LIN {X 0,Y 297.522,Z 437.012,A -85,B 0,C 180,E1 -16370.483,E2 -16370.483} C_VEL
LIN {X 0,Y 297.104,Z 437.216,A -85,B 0,C 180,E1 -16373.208,E2 -16373.208} C_VEL
LIN {X 0,Y 296.911,Z 436.192,A -85,B 0,C 180,E1 -16375.928,E2 -16375.928} C_VEL
LIN {X 0,Y 296.872,Z 433.944,A -85,B 0,C 180,E1 -16378.644,E2 -16378.644} C_VEL
LIN {X 0,Y 296.926,Z 430.435,A -85,B 0,C 180,E1 -16381.357,E2 -16381.357} C_VEL
LIN {X 0,Y 297.311,Z 426.96,A -85,B 0,C 180,E1 -16383.388,E2 -16383.388} C_VEL
LIN {X 0,Y 297.857,Z 421.058,A -85,B 0,C 180,E1 -16386.095,E2 -16386.095} C_VEL
LIN {X 0,Y 298.455,Z 414.521,A -85,B 0,C 180,E1 -16388.499,E2 -16388.499} C_VEL
LIN {X 0,Y 299.541,Z 405.637,A -85,B 0,C 180,E1 -16391.161,E2 -16391.161} C_VEL
LIN {X 0,Y 300.946,Z 396.119,A -85,B 0,C 180,E1 -16393.505,E2 -16393.505} C_VEL
LIN {X 0,Y 302.502,Z 384.733,A -85,B 0,C 180,E1 -16395.842,E2 -16395.842} C_VEL
LIN {X 0,Y 304.428,Z 372.118,A -85,B 0,C 180,E1 -16397.986,E2 -16397.986} C_VEL
LIN {X 0,Y 306.235,Z 358.613,A -85,B 0,C 180,E1 -16399.902,E2 -16399.902} C_VEL
LIN {X 0,Y 308.168,Z 344.283,A -85,B 0,C 180,E1 -16401.577,E2 -16401.577} C_VEL
LIN {X 0,Y 309.992,Z 329.479,A -85,B 0,C 180,E1 -16402.99,E2 -16402.99} C_VEL
LIN {X 0,Y 309.934,Z 327.134,A -85,B 0,C 180,E1 -16403.209,E2 -16403.209} C_VEL
LIN {X 0,Y 306.166,Z 312.141,A -85,B 0,C 180,E1 -16404.665,E2 -16404.665} C_VEL
LIN {X 0,Y 301.591,Z 296.002,A -85,B 0,C 180,E1 -16406.023,E2 -16406.023} C_VEL
LIN {X 0,Y 297.601,Z 283.041,A -85,B 0,C 180,E1 -16407.007,E2 -16407.007} C_VEL
LIN {X 0,Y 297.87,Z 283.005,A -85,B 0,C 180,E1 -16409.702,E2 -16409.702} C_VEL
LIN {X 0,Y 298.165,Z 282.969,A -85,B 0,C 180,E1 -16412.829,E2 -16412.829} C_VEL
LIN {X 0,Y 298.368,Z 282.942,A -85,B 0,C 180,E1 -16416.077,E2 -16416.077} C_VEL
LIN {X 0,Y 298.403,Z 282.94,A -85,B 0,C 180,E1 -16419.488,E2 -16419.488} C_VEL
LIN {X 0,Y 298.401,Z 282.942,A -85,B 0,C 180,E1 -16423.103,E2 -16423.103} C_VEL
LIN {X 0,Y 298.405,Z 282.941,A -85,B 0,C 180,E1 -16426.921,E2 -16426.921} C_VEL
LIN {X 0,Y 298.401,Z 282.941,A -85,B 0,C 180,E1 -16431.007,E2 -16431.007} C_VEL
LIN {X 0,Y 298.421,Z 282.935,A -85,B 0,C 180,E1 -16433.93,E2 -16433.93} C_VEL
LIN {X 0,Y 298.396,Z 282.938,A -85,B 0,C 180,E1 -16437.984,E2 -16437.984} C_VEL
LIN {X 0,Y 298.46,Z 282.93,A -85,B 0,C 180,E1 -16441.904,E2 -16441.904} C_VEL
LIN {X 0,Y 298.484,Z 282.928,A -85,B 0,C 180,E1 -16444.924,E2 -16444.924} C_VEL
LIN {X 0,Y 298.436,Z 282.933,A -85,B 0,C 180,E1 -16449.314,E2 -16449.314} C_VEL
LIN {X 0,Y 298.538,Z 282.924,A -85,B 0,C 180,E1 -16452.179,E2 -16452.179} C_VEL
LIN {X 0,Y 298.597,Z 282.913,A -85,B 0,C 180,E1 -16454.995,E2 -16454.995} C_VEL
LIN {X 0,Y 298.594,Z 282.913,A -85,B 0,C 180,E1 -16459.147,E2 -16459.147} C_VEL
LIN {X 0,Y 298.701,Z 282.902,A -85,B 0,C 180,E1 -16461.884,E2 -16461.884} C_VEL
LIN {X 0,Y 298.637,Z 282.909,A -85,B 0,C 180,E1 -16464.599,E2 -16464.599} C_VEL
LIN {X 0,Y 298.923,Z 282.872,A -85,B 0,C 180,E1 -16468.653,E2 -16468.653} C_VEL
LIN {X 0,Y 298.922,Z 282.872,A -85,B 0,C 180,E1 -16471.347,E2 -16471.347} C_VEL
LIN {X 0,Y 298.643,Z 282.909,A -85,B 0,C 180,E1 -16475.401,E2 -16475.401} C_VEL
LIN {X 0,Y 298.713,Z 282.9,A -85,B 0,C 180,E1 -16478.115,E2 -16478.115} C_VEL
LIN {X 0,Y 298.553,Z 282.919,A -85,B 0,C 180,E1 -16482.232,E2 -16482.232} C_VEL
LIN {X 0,Y 298.609,Z 282.913,A -85,B 0,C 180,E1 -16485.209,E2 -16485.209} C_VEL
LIN {X 0,Y 298.543,Z 282.921,A -85,B 0,C 180,E1 -16489.243,E2 -16489.243} C_VEL
LIN {X 0,Y 298.461,Z 282.933,A -85,B 0,C 180,E1 -16493.598,E2 -16493.598} C_VEL
LIN {X 0,Y 298.488,Z 282.926,A -85,B 0,C 180,E1 -16496.575,E2 -16496.575} C_VEL
LIN {X 0,Y 298.42,Z 282.937,A -85,B 0,C 180,E1 -16499.641,E2 -16499.641} C_VEL
LIN {X 0,Y 298.398,Z 282.939,A -85,B 0,C 180,E1 -16502.8,E2 -16502.8} C_VEL
LIN {X 0,Y 298.431,Z 282.935,A -85,B 0,C 180,E1 -16506.803,E2 -16506.803} C_VEL
LIN {X 0,Y 298.376,Z 282.942,A -85,B 0,C 180,E1 -16509.492,E2 -16509.492} C_VEL
LIN {X 0,Y 298.374,Z 282.945,A -85,B 0,C 180,E1 -16513.097,E2 -16513.097} C_VEL
LIN {X 0,Y 298.406,Z 282.942,A -85,B 0,C 180,E1 -16516.921,E2 -16516.921} C_VEL
LIN {X 0,Y 298.402,Z 282.94,A -85,B 0,C 180,E1 -16521.007,E2 -16521.007} C_VEL
LIN {X 0,Y 298.421,Z 282.935,A -85,B 0,C 180,E1 -16523.93,E2 -16523.93} C_VEL
LIN {X 0,Y 298.397,Z 282.938,A -85,B 0,C 180,E1 -16527.984,E2 -16527.984} C_VEL
LIN {X 0,Y 298.461,Z 282.93,A -85,B 0,C 180,E1 -16531.904,E2 -16531.904} C_VEL
LIN {X 0,Y 298.485,Z 282.928,A -85,B 0,C 180,E1 -16534.924,E2 -16534.924} C_VEL
LIN {X 0,Y 298.444,Z 282.932,A -85,B 0,C 180,E1 -16539.314,E2 -16539.314} C_VEL
LIN {X 0,Y 298.542,Z 282.923,A -85,B 0,C 180,E1 -16542.179,E2 -16542.179} C_VEL
LIN {X 0,Y 298.597,Z 282.912,A -85,B 0,C 180,E1 -16544.995,E2 -16544.995} C_VEL
LIN {X 0,Y 298.587,Z 282.914,A -85,B 0,C 180,E1 -16549.146,E2 -16549.146} C_VEL
LIN {X 0,Y 298.702,Z 282.902,A -85,B 0,C 180,E1 -16551.884,E2 -16551.884} C_VEL
LIN {X 0,Y 298.639,Z 282.909,A -85,B 0,C 180,E1 -16554.598,E2 -16554.598} C_VEL
LIN {X 0,Y 298.924,Z 282.873,A -85,B 0,C 180,E1 -16558.652,E2 -16558.652} C_VEL
LIN {X 0,Y 298.922,Z 282.872,A -85,B 0,C 180,E1 -16561.347,E2 -16561.347} C_VEL
LIN {X 0,Y 298.854,Z 282.878,A -85,B 0,C 180,E1 -16562.103,E2 -16562.103} C_VEL
LIN {X 0,Y 298.135,Z 282.971,A -85,B 0,C 180,E1 -16563.226,E2 -16563.226} C_VEL
LIN {X 0,Y 295.21,Z 283.335,A -85,B 0,C 180,E1 -16565.053,E2 -16565.053} C_VEL
LIN {X 0,Y 292.761,Z 283.64,A -85,B 0,C 180,E1 -16566.536,E2 -16566.536} C_VEL
LIN {X 0,Y 291.726,Z 283.772,A -85,B 0,C 180,E1 -16567.686,E2 -16567.686} C_VEL
LIN {X 0,Y 291.649,Z 283.777,A -85,B 0,C 180,E1 -16568.075,E2 -16568.075} C_VEL
LIN {X 0,Y 291.521,Z 283.794,A -85,B 0,C 180,E1 -16572.531,E2 -16572.531} C_VEL
LIN {X 0,Y 291.558,Z 283.792,A -85,B 0,C 180,E1 -16575.376,E2 -16575.376} C_VEL
LIN {X 0,Y 291.453,Z 283.805,A -85,B 0,C 180,E1 -16579.874,E2 -16579.874} C_VEL
LIN {X 0,Y 291.366,Z 283.815,A -85,B 0,C 180,E1 -16584.208,E2 -16584.208} C_VEL
LIN {X 0,Y 291.355,Z 283.819,A -85,B 0,C 180,E1 -16587.278,E2 -16587.278} C_VEL
LIN {X 0,Y 291.391,Z 283.877,A -85,B 0,C 180,E1 -16589.079,E2 -16589.079} C_VEL
LIN {X 0,Y 291.971,Z 287.579,A -85,B 0,C 180,E1 -16592.596,E2 -16592.596} C_VEL
LIN {X 0,Y 292.796,Z 292.36,A -85,B 0,C 180,E1 -16596.875,E2 -16596.875} C_VEL
LIN {X 0,Y 293.772,Z 297.435,A -85,B 0,C 180,E1 -16601.139,E2 -16601.139} C_VEL
LIN {X 0,Y 294.512,Z 301.385,A -85,B 0,C 180,E1 -16604.283,E2 -16604.283} C_VEL
LIN {X 0,Y 294.887,Z 304.002,A -85,B 0,C 180,E1 -16606.278,E2 -16606.278} C_VEL
LIN {X 0,Y 294.882,Z 306.534,A -85,B 0,C 180,E1 -16608.138,E2 -16608.138} C_VEL
LIN {X 0,Y 294.127,Z 311.482,A -85,B 0,C 180,E1 -16611.592,E2 -16611.592} C_VEL
LIN {X 0,Y 293.063,Z 317.71,A -85,B 0,C 180,E1 -16615.796,E2 -16615.796} C_VEL
LIN {X 0,Y 297.438,Z 336.476,A -85,B 0,C 180,E1 -16617.196,E2 -16617.196} C_VEL
LIN {X 0,Y 300.916,Z 353.108,A -85,B 0,C 180,E1 -16618.669,E2 -16618.669} C_VEL
LIN {X 0,Y 303.835,Z 368.951,A -85,B 0,C 180,E1 -16620.322,E2 -16620.322} C_VEL
LIN {X 0,Y 305.212,Z 379.329,A -85,B 0,C 180,E1 -16621.521,E2 -16621.521} C_VEL
LIN {X 0,Y 302.653,Z 392.931,A -85,B 0,C 180,E1 -16623.075,E2 -16623.075} C_VEL
LIN {X 0,Y 300.081,Z 405.907,A -85,B 0,C 180,E1 -16624.881,E2 -16624.881} C_VEL
LIN {X 0,Y 297.678,Z 417.982,A -85,B 0,C 180,E1 -16626.913,E2 -16626.913} C_VEL
LIN {X 0,Y 295.517,Z 428.788,A -85,B 0,C 180,E1 -16629.1,E2 -16629.1} C_VEL
LIN {X 0,Y 293.557,Z 438.678,A -85,B 0,C 180,E1 -16631.505,E2 -16631.505} C_VEL
LIN {X 0,Y 292.031,Z 447.172,A -85,B 0,C 180,E1 -16634.005,E2 -16634.005} C_VEL
LIN {X 0,Y 290.853,Z 454.729,A -85,B 0,C 180,E1 -16636.729,E2 -16636.729} C_VEL
LIN {X 0,Y 290.093,Z 460.885,A -85,B 0,C 180,E1 -16639.531,E2 -16639.531} C_VEL
LIN {X 0,Y 289.749,Z 465.59,A -85,B 0,C 180,E1 -16642.333,E2 -16642.333} C_VEL
LIN {X 0,Y 289.648,Z 468.242,A -85,B 0,C 180,E1 -16644.43,E2 -16644.43} C_VEL
LIN {X 0,Y 289.543,Z 470.632,A -85,B 0,C 180,E1 -16647.217,E2 -16647.217} C_VEL
LIN {X 0,Y 289.657,Z 471.738,A -85,B 0,C 180,E1 -16650,E2 -16650} C_VEL
LIN {X 0,Y 289.539,Z 471.604,A -85,B 0,C 180,E1 -16652.783,E2 -16652.783} C_VEL
LIN {X 0,Y 289.585,Z 470.189,A -85,B 0,C 180,E1 -16655.712,E2 -16655.712} C_VEL
LIN {X 0,Y 289.712,Z 467.815,A -85,B 0,C 180,E1 -16658.369,E2 -16658.369} C_VEL
LIN {X 0,Y 290.177,Z 464.167,A -85,B 0,C 180,E1 -16661.172,E2 -16661.172} C_VEL
LIN {X 0,Y 291.19,Z 459.315,A -85,B 0,C 180,E1 -16663.967,E2 -16663.967} C_VEL
LIN {X 0,Y 292.734,Z 453.256,A -85,B 0,C 180,E1 -16666.744,E2 -16666.744} C_VEL
LIN {X 0,Y 295.205,Z 444.929,A -85,B 0,C 180,E1 -16669.831,E2 -16669.831} C_VEL
LIN {X 0,Y 298.479,Z 434.898,A -85,B 0,C 180,E1 -16672.862,E2 -16672.862} C_VEL
LIN {X 0,Y 302.294,Z 424.35,A -85,B 0,C 180,E1 -16675.474,E2 -16675.474} C_VEL
LIN {X 0,Y 306.87,Z 412.141,A -85,B 0,C 180,E1 -16678.002,E2 -16678.002} C_VEL
LIN {X 0,Y 311.549,Z 399.815,A -85,B 0,C 180,E1 -16680.127,E2 -16680.127} C_VEL
LIN {X 0,Y 316.135,Z 387.773,A -85,B 0,C 180,E1 -16681.878,E2 -16681.878} C_VEL
LIN {X 0,Y 318.826,Z 373.737,A -85,B 0,C 180,E1 -16684.272,E2 -16684.272} C_VEL
LIN {X 0,Y 319.606,Z 365.662,A -85,B 0,C 180,E1 -16685.875,E2 -16685.875} C_VEL
LIN {X 0,Y 319.866,Z 359.589,A -85,B 0,C 180,E1 -16687.285,E2 -16687.285} C_VEL
LIN {X 0,Y 319.968,Z 353.405,A -85,B 0,C 180,E1 -16689.036,E2 -16689.036} C_VEL
LIN {X 0,Y 320.152,Z 347.624,A -85,B 0,C 180,E1 -16691.191,E2 -16691.191} C_VEL
LIN {X 0,Y 320.329,Z 344.817,A -85,B 0,C 180,E1 -16692.855,E2 -16692.855} C_VEL
LIN {X 0,Y 320.856,Z 342.981,A -85,B 0,C 180,E1 -16694.502,E2 -16694.502} C_VEL
LIN {X 0,Y 321.371,Z 342.809,A -85,B 0,C 180,E1 -16696.193,E2 -16696.193} C_VEL
LIN {X 0,Y 322.187,Z 343.704,A -85,B 0,C 180,E1 -16697.873,E2 -16697.873} C_VEL
LIN {X 0,Y 323.235,Z 345.85,A -85,B 0,C 180,E1 -16699.552,E2 -16699.552} C_VEL
LIN {X 0,Y 324.353,Z 349.259,A -85,B 0,C 180,E1 -16701.265,E2 -16701.265} C_VEL
LIN {X 0,Y 325.411,Z 354.292,A -85,B 0,C 180,E1 -16703.045,E2 -16703.045} C_VEL
LIN {X 0,Y 325.075,Z 355.962,A -85,B 0,C 180,E1 -16703.336,E2 -16703.336} C_VEL
LIN {X 0,Y 319.824,Z 369.536,A -85,B 0,C 180,E1 -16705.157,E2 -16705.157} C_VEL
LIN {X 0,Y 315.395,Z 380.551,A -85,B 0,C 180,E1 -16706.912,E2 -16706.912} C_VEL
LIN {X 0,Y 310.561,Z 392.234,A -85,B 0,C 180,E1 -16709.145,E2 -16709.145} C_VEL
LIN {X 0,Y 306.14,Z 402.677,A -85,B 0,C 180,E1 -16711.553,E2 -16711.553} C_VEL
LIN {X 0,Y 302.648,Z 410.832,A -85,B 0,C 180,E1 -16713.819,E2 -16713.819} C_VEL
LIN {X 0,Y 299.236,Z 418.664,A -85,B 0,C 180,E1 -16716.468,E2 -16716.468} C_VEL
LIN {X 0,Y 296.458,Z 425.035,A -85,B 0,C 180,E1 -16719.17,E2 -16719.17} C_VEL
LIN {X 0,Y 294.256,Z 430.053,A -85,B 0,C 180,E1 -16721.911,E2 -16721.911} C_VEL
LIN {X 0,Y 292.632,Z 433.797,A -85,B 0,C 180,E1 -16724.682,E2 -16724.682} C_VEL
LIN {X 0,Y 291.305,Z 436.315,A -85,B 0,C 180,E1 -16727.46,E2 -16727.46} C_VEL
LIN {X 0,Y 290.494,Z 437.641,A -85,B 0,C 180,E1 -16730.25,E2 -16730.25} C_VEL
LIN {X 0,Y 290.037,Z 437.758,A -85,B 0,C 180,E1 -16733.041,E2 -16733.041} C_VEL
LIN {X 0,Y 289.846,Z 436.635,A -85,B 0,C 180,E1 -16735.829,E2 -16735.829} C_VEL
LIN {X 0,Y 289.777,Z 434.29,A -85,B 0,C 180,E1 -16738.611,E2 -16738.611} C_VEL
LIN {X 0,Y 289.833,Z 430.688,A -85,B 0,C 180,E1 -16741.39,E2 -16741.39} C_VEL
LIN {X 0,Y 290.263,Z 425.732,A -85,B 0,C 180,E1 -16744.166,E2 -16744.166} C_VEL
LIN {X 0,Y 290.811,Z 421.095,A -85,B 0,C 180,E1 -16746.244,E2 -16746.244} C_VEL
LIN {X 0,Y 291.511,Z 413.513,A -85,B 0,C 180,E1 -16749.016,E2 -16749.016} C_VEL
LIN {X 0,Y 292.57,Z 405.45,A -85,B 0,C 180,E1 -16751.431,E2 -16751.431} C_VEL
LIN {X 0,Y 294,Z 395.835,A -85,B 0,C 180,E1 -16753.831,E2 -16753.831} C_VEL
LIN {X 0,Y 295.403,Z 386.14,A -85,B 0,C 180,E1 -16755.879,E2 -16755.879} C_VEL
LIN {X 0,Y 297.314,Z 373.683,A -85,B 0,C 180,E1 -16758.075,E2 -16758.075} C_VEL
LIN {X 0,Y 299.168,Z 360.601,A -85,B 0,C 180,E1 -16760.002,E2 -16760.002} C_VEL
LIN {X 0,Y 300.887,Z 347.794,A -85,B 0,C 180,E1 -16761.585,E2 -16761.585} C_VEL
LIN {X 0,Y 302.794,Z 333.32,A -85,B 0,C 180,E1 -16763.059,E2 -16763.059} C_VEL
LIN {X 0,Y 303.223,Z 329.818,A -85,B 0,C 180,E1 -16763.376,E2 -16763.376} C_VEL
LIN {X 0,Y 301.005,Z 319.776,A -85,B 0,C 180,E1 -16764.412,E2 -16764.412} C_VEL
LIN {X 0,Y 296.81,Z 304.173,A -85,B 0,C 180,E1 -16765.87,E2 -16765.87} C_VEL
LIN {X 0,Y 292.073,Z 288.316,A -85,B 0,C 180,E1 -16767.147,E2 -16767.147} C_VEL
LIN {X 0,Y 290.628,Z 283.91,A -85,B 0,C 180,E1 -16767.499,E2 -16767.499} C_VEL
LIN {X 0,Y 290.886,Z 283.874,A -85,B 0,C 180,E1 -16770.489,E2 -16770.489} C_VEL
LIN {X 0,Y 291.163,Z 283.84,A -85,B 0,C 180,E1 -16773.723,E2 -16773.723} C_VEL
LIN {X 0,Y 291.353,Z 283.82,A -85,B 0,C 180,E1 -16777.247,E2 -16777.247} C_VEL
LIN {X 0,Y 291.335,Z 283.821,A -85,B 0,C 180,E1 -16780.643,E2 -16780.643} C_VEL
LIN {X 0,Y 291.292,Z 283.824,A -85,B 0,C 180,E1 -16784.402,E2 -16784.402} C_VEL
LIN {X 0,Y 291.33,Z 283.819,A -85,B 0,C 180,E1 -16788.404,E2 -16788.404} C_VEL
LIN {X 0,Y 291.35,Z 283.818,A -85,B 0,C 180,E1 -16791.158,E2 -16791.158} C_VEL
LIN {X 0,Y 291.364,Z 283.818,A -85,B 0,C 180,E1 -16794.626,E2 -16794.626} C_VEL
LIN {X 0,Y 291.373,Z 283.813,A -85,B 0,C 180,E1 -16797.951,E2 -16797.951} C_VEL
LIN {X 0,Y 291.38,Z 283.813,A -85,B 0,C 180,E1 -16801.158,E2 -16801.158} C_VEL
LIN {X 0,Y 291.414,Z 283.81,A -85,B 0,C 180,E1 -16804.272,E2 -16804.272} C_VEL
LIN {X 0,Y 291.374,Z 283.812,A -85,B 0,C 180,E1 -16807.299,E2 -16807.299} C_VEL
LIN {X 0,Y 291.461,Z 283.806,A -85,B 0,C 180,E1 -16810.27,E2 -16810.27} C_VEL
LIN {X 0,Y 291.558,Z 283.791,A -85,B 0,C 180,E1 -16814.624,E2 -16814.624} C_VEL
LIN {X 0,Y 291.538,Z 283.793,A -85,B 0,C 180,E1 -16818.881,E2 -16818.881} C_VEL
LIN {X 0,Y 291.654,Z 283.779,A -85,B 0,C 180,E1 -16821.687,E2 -16821.687} C_VEL
LIN {X 0,Y 291.606,Z 283.785,A -85,B 0,C 180,E1 -16824.468,E2 -16824.468} C_VEL
LIN {X 0,Y 291.889,Z 283.749,A -85,B 0,C 180,E1 -16828.62,E2 -16828.62} C_VEL
LIN {X 0,Y 291.888,Z 283.749,A -85,B 0,C 180,E1 -16831.38,E2 -16831.38} C_VEL
LIN {X 0,Y 291.612,Z 283.785,A -85,B 0,C 180,E1 -16835.532,E2 -16835.532} C_VEL
LIN {X 0,Y 291.676,Z 283.774,A -85,B 0,C 180,E1 -16838.918,E2 -16838.918} C_VEL
LIN {X 0,Y 291.525,Z 283.796,A -85,B 0,C 180,E1 -16843.95,E2 -16843.95} C_VEL
LIN {X 0,Y 291.49,Z 283.798,A -85,B 0,C 180,E1 -16846.818,E2 -16846.818} C_VEL
LIN {X 0,Y 291.454,Z 283.805,A -85,B 0,C 180,E1 -16849.875,E2 -16849.875} C_VEL
LIN {X 0,Y 291.403,Z 283.809,A -85,B 0,C 180,E1 -16854.205,E2 -16854.205} C_VEL
LIN {X 0,Y 291.422,Z 283.81,A -85,B 0,C 180,E1 -16857.272,E2 -16857.272} C_VEL
LIN {X 0,Y 291.337,Z 283.817,A -85,B 0,C 180,E1 -16860.437,E2 -16860.437} C_VEL
LIN {X 0,Y 291.347,Z 283.816,A -85,B 0,C 180,E1 -16863.698,E2 -16863.698} C_VEL
LIN {X 0,Y 291.362,Z 283.818,A -85,B 0,C 180,E1 -16867.25,E2 -16867.25} C_VEL
LIN {X 0,Y 291.303,Z 283.823,A -85,B 0,C 180,E1 -16870.648,E2 -16870.648} C_VEL
LIN {X 0,Y 291.284,Z 283.824,A -85,B 0,C 180,E1 -16874.404,E2 -16874.404} C_VEL
LIN {X 0,Y 291.33,Z 283.819,A -85,B 0,C 180,E1 -16878.404,E2 -16878.404} C_VEL
LIN {X 0,Y 291.351,Z 283.817,A -85,B 0,C 180,E1 -16881.158,E2 -16881.158} C_VEL
LIN {X 0,Y 291.364,Z 283.817,A -85,B 0,C 180,E1 -16884.626,E2 -16884.626} C_VEL
LIN {X 0,Y 291.374,Z 283.812,A -85,B 0,C 180,E1 -16887.951,E2 -16887.951} C_VEL
LIN {X 0,Y 291.38,Z 283.813,A -85,B 0,C 180,E1 -16891.158,E2 -16891.158} C_VEL
LIN {X 0,Y 291.415,Z 283.81,A -85,B 0,C 180,E1 -16894.271,E2 -16894.271} C_VEL
LIN {X 0,Y 291.378,Z 283.811,A -85,B 0,C 180,E1 -16897.299,E2 -16897.299} C_VEL
LIN {X 0,Y 291.461,Z 283.805,A -85,B 0,C 180,E1 -16900.27,E2 -16900.27} C_VEL
LIN {X 0,Y 291.559,Z 283.791,A -85,B 0,C 180,E1 -16904.624,E2 -16904.624} C_VEL
LIN {X 0,Y 291.533,Z 283.793,A -85,B 0,C 180,E1 -16908.88,E2 -16908.88} C_VEL
LIN {X 0,Y 291.655,Z 283.779,A -85,B 0,C 180,E1 -16911.687,E2 -16911.687} C_VEL
LIN {X 0,Y 291.608,Z 283.785,A -85,B 0,C 180,E1 -16914.468,E2 -16914.468} C_VEL
LIN {X 0,Y 291.89,Z 283.749,A -85,B 0,C 180,E1 -16918.62,E2 -16918.62} C_VEL
LIN {X 0,Y 291.817,Z 283.754,A -85,B 0,C 180,E1 -16922.084,E2 -16922.084} C_VEL
LIN {X 0,Y 291.692,Z 283.773,A -85,B 0,C 180,E1 -16926.919,E2 -16926.919} C_VEL
LIN {X 0,Y 291.649,Z 283.777,A -85,B 0,C 180,E1 -16928.075,E2 -16928.075} C_VEL
LIN {X 0,Y 290.975,Z 283.865,A -85,B 0,C 180,E1 -16929.227,E2 -16929.227} C_VEL
LIN {X 0,Y 288.039,Z 284.228,A -85,B 0,C 180,E1 -16931.099,E2 -16931.099} C_VEL
LIN {X 0,Y 285.565,Z 284.536,A -85,B 0,C 180,E1 -16932.619,E2 -16932.619} C_VEL
LIN {X 0,Y 284.541,Z 284.668,A -85,B 0,C 180,E1 -16933.8,E2 -16933.8} C_VEL
LIN {X 0,Y 284.478,Z 284.672,A -85,B 0,C 180,E1 -16934.2,E2 -16934.2} C_VEL
LIN {X 0,Y 284.428,Z 284.679,A -85,B 0,C 180,E1 -16937.248,E2 -16937.248} C_VEL
LIN {X 0,Y 284.383,Z 284.684,A -85,B 0,C 180,E1 -16940.242,E2 -16940.242} C_VEL
LIN {X 0,Y 284.326,Z 284.693,A -85,B 0,C 180,E1 -16943.854,E2 -16943.854} C_VEL
LIN {X 0,Y 284.288,Z 284.697,A -85,B 0,C 180,E1 -16948.015,E2 -16948.015} C_VEL
LIN {X 0,Y 284.339,Z 284.925,A -85,B 0,C 180,E1 -16948.815,E2 -16948.815} C_VEL
LIN {X 0,Y 284.736,Z 287.382,A -85,B 0,C 180,E1 -16951.22,E2 -16951.22} C_VEL
LIN {X 0,Y 285.32,Z 290.884,A -85,B 0,C 180,E1 -16954.509,E2 -16954.509} C_VEL
LIN {X 0,Y 286.067,Z 295.003,A -85,B 0,C 180,E1 -16958.171,E2 -16958.171} C_VEL
LIN {X 0,Y 287.174,Z 300.469,A -85,B 0,C 180,E1 -16962.761,E2 -16962.761} C_VEL
LIN {X 0,Y 287.807,Z 304.547,A -85,B 0,C 180,E1 -16965.979,E2 -16965.979} C_VEL
LIN {X 0,Y 287.738,Z 308.254,A -85,B 0,C 180,E1 -16968.74,E2 -16968.74} C_VEL
LIN {X 0,Y 286.882,Z 313.173,A -85,B 0,C 180,E1 -16972.233,E2 -16972.233} C_VEL
LIN {X 0,Y 286.134,Z 317.418,A -85,B 0,C 180,E1 -16975.167,E2 -16975.167} C_VEL
LIN {X 0,Y 290.424,Z 336.297,A -85,B 0,C 180,E1 -16976.602,E2 -16976.602} C_VEL
LIN {X 0,Y 293.616,Z 351.694,A -85,B 0,C 180,E1 -16978.002,E2 -16978.002} C_VEL
LIN {X 0,Y 296.363,Z 366.3,A -85,B 0,C 180,E1 -16979.541,E2 -16979.541} C_VEL
LIN {X 0,Y 298.38,Z 379.834,A -85,B 0,C 180,E1 -16981.151,E2 -16981.151} C_VEL
LIN {X 0,Y 295.709,Z 393.513,A -85,B 0,C 180,E1 -16982.773,E2 -16982.773} C_VEL
LIN {X 0,Y 293.095,Z 406.291,A -85,B 0,C 180,E1 -16984.62,E2 -16984.62} C_VEL
LIN {X 0,Y 290.556,Z 418.734,A -85,B 0,C 180,E1 -16986.801,E2 -16986.801} C_VEL
LIN {X 0,Y 288.475,Z 428.902,A -85,B 0,C 180,E1 -16988.94,E2 -16988.94} C_VEL
LIN {X 0,Y 286.47,Z 438.685,A -85,B 0,C 180,E1 -16991.402,E2 -16991.402} C_VEL
LIN {X 0,Y 284.966,Z 446.873,A -85,B 0,C 180,E1 -16993.891,E2 -16993.891} C_VEL
LIN {X 0,Y 283.877,Z 453.675,A -85,B 0,C 180,E1 -16996.397,E2 -16996.397} C_VEL
LIN {X 0,Y 283.052,Z 459.958,A -85,B 0,C 180,E1 -16999.268,E2 -16999.268} C_VEL
LIN {X 0,Y 282.685,Z 464.781,A -85,B 0,C 180,E1 -17002.141,E2 -17002.141} C_VEL
LIN {X 0,Y 282.589,Z 467.536,A -85,B 0,C 180,E1 -17004.291,E2 -17004.291} C_VEL
LIN {X 0,Y 282.564,Z 468.927,A -85,B 0,C 180,E1 -17005.721,E2 -17005.721} C_VEL
LIN {X 0,Y 282.525,Z 470.742,A -85,B 0,C 180,E1 -17008.575,E2 -17008.575} C_VEL
LIN {X 0,Y 282.577,Z 471.191,A -85,B 0,C 180,E1 -17010,E2 -17010} C_VEL
LIN {X 0,Y 282.465,Z 471.165,A -85,B 0,C 180,E1 -17012.852,E2 -17012.852} C_VEL
LIN {X 0,Y 282.486,Z 469.962,A -85,B 0,C 180,E1 -17015.711,E2 -17015.711} C_VEL
LIN {X 0,Y 282.637,Z 467.592,A -85,B 0,C 180,E1 -17018.58,E2 -17018.58} C_VEL
LIN {X 0,Y 283.403,Z 462.998,A -85,B 0,C 180,E1 -17022.169,E2 -17022.169} C_VEL
LIN {X 0,Y 284.617,Z 458.033,A -85,B 0,C 180,E1 -17025.027,E2 -17025.027} C_VEL
LIN {X 0,Y 286.395,Z 451.846,A -85,B 0,C 180,E1 -17027.863,E2 -17027.863} C_VEL
LIN {X 0,Y 289.25,Z 443.425,A -85,B 0,C 180,E1 -17031.001,E2 -17031.001} C_VEL
LIN {X 0,Y 292.436,Z 434.528,A -85,B 0,C 180,E1 -17033.736,E2 -17033.736} C_VEL
LIN {X 0,Y 297.082,Z 422.82,A -85,B 0,C 180,E1 -17036.71,E2 -17036.71} C_VEL
LIN {X 0,Y 302.113,Z 410.629,A -85,B 0,C 180,E1 -17039.243,E2 -17039.243} C_VEL
LIN {X 0,Y 308.017,Z 396.506,A -85,B 0,C 180,E1 -17041.654,E2 -17041.654} C_VEL
LIN {X 0,Y 310.492,Z 390.627,A -85,B 0,C 180,E1 -17042.528,E2 -17042.528} C_VEL
LIN {X 0,Y 313.836,Z 377.026,A -85,B 0,C 180,E1 -17044.961,E2 -17044.961} C_VEL
LIN {X 0,Y 315.068,Z 368.457,A -85,B 0,C 180,E1 -17046.784,E2 -17046.784} C_VEL
LIN {X 0,Y 315.671,Z 361.687,A -85,B 0,C 180,E1 -17048.564,E2 -17048.564} C_VEL
LIN {X 0,Y 316.025,Z 356.796,A -85,B 0,C 180,E1 -17050.16,E2 -17050.16} C_VEL
LIN {X 0,Y 316.482,Z 352.965,A -85,B 0,C 180,E1 -17051.775,E2 -17051.775} C_VEL
LIN {X 0,Y 316.888,Z 350.382,A -85,B 0,C 180,E1 -17053.435,E2 -17053.435} C_VEL
LIN {X 0,Y 317.496,Z 348.996,A -85,B 0,C 180,E1 -17055.101,E2 -17055.101} C_VEL
LIN {X 0,Y 318.062,Z 349.233,A -85,B 0,C 180,E1 -17056.818,E2 -17056.818} C_VEL
LIN {X 0,Y 319.212,Z 351.409,A -85,B 0,C 180,E1 -17059.181,E2 -17059.181} C_VEL
LIN {X 0,Y 320.123,Z 354.653,A -85,B 0,C 180,E1 -17060.946,E2 -17060.946} C_VEL
LIN {X 0,Y 320.639,Z 357.726,A -85,B 0,C 180,E1 -17062.141,E2 -17062.141} C_VEL
LIN {X 0,Y 320.308,Z 359.633,A -85,B 0,C 180,E1 -17062.584,E2 -17062.584} C_VEL
LIN {X 0,Y 314.572,Z 373.129,A -85,B 0,C 180,E1 -17064.488,E2 -17064.488} C_VEL
LIN {X 0,Y 308.518,Z 386.788,A -85,B 0,C 180,E1 -17066.858,E2 -17066.858} C_VEL
LIN {X 0,Y 303.176,Z 398.386,A -85,B 0,C 180,E1 -17069.337,E2 -17069.337} C_VEL
LIN {X 0,Y 298.558,Z 408.255,A -85,B 0,C 180,E1 -17071.914,E2 -17071.914} C_VEL
LIN {X 0,Y 294.627,Z 416.545,A -85,B 0,C 180,E1 -17074.573,E2 -17074.573} C_VEL
LIN {X 0,Y 291.311,Z 423.387,A -85,B 0,C 180,E1 -17077.294,E2 -17077.294} C_VEL
LIN {X 0,Y 288.72,Z 428.843,A -85,B 0,C 180,E1 -17080.075,E2 -17080.075} C_VEL
LIN {X 0,Y 286.393,Z 433.408,A -85,B 0,C 180,E1 -17083.148,E2 -17083.148} C_VEL
LIN {X 0,Y 284.968,Z 436.04,A -85,B 0,C 180,E1 -17085.722,E2 -17085.722} C_VEL
LIN {X 0,Y 283.88,Z 437.817,A -85,B 0,C 180,E1 -17088.577,E2 -17088.577} C_VEL
LIN {X 0,Y 283.192,Z 438.42,A -85,B 0,C 180,E1 -17091.437,E2 -17091.437} C_VEL
LIN {X 0,Y 282.876,Z 437.82,A -85,B 0,C 180,E1 -17094.297,E2 -17094.297} C_VEL
LIN {X 0,Y 282.697,Z 436.003,A -85,B 0,C 180,E1 -17097.15,E2 -17097.15} C_VEL
LIN {X 0,Y 282.683,Z 432.923,A -85,B 0,C 180,E1 -17100,E2 -17100} C_VEL
LIN {X 0,Y 282.914,Z 428.551,A -85,B 0,C 180,E1 -17102.848,E2 -17102.848} C_VEL
LIN {X 0,Y 283.589,Z 422.801,A -85,B 0,C 180,E1 -17105.689,E2 -17105.689} C_VEL
LIN {X 0,Y 284.231,Z 415.515,A -85,B 0,C 180,E1 -17108.532,E2 -17108.532} C_VEL
LIN {X 0,Y 285.404,Z 406.505,A -85,B 0,C 180,E1 -17111.362,E2 -17111.362} C_VEL
LIN {X 0,Y 286.868,Z 396.979,A -85,B 0,C 180,E1 -17113.82,E2 -17113.82} C_VEL
LIN {X 0,Y 288.526,Z 385.599,A -85,B 0,C 180,E1 -17116.268,E2 -17116.268} C_VEL
LIN {X 0,Y 290.51,Z 373.015,A -85,B 0,C 180,E1 -17118.513,E2 -17118.513} C_VEL
LIN {X 0,Y 292.447,Z 359.583,A -85,B 0,C 180,E1 -17120.514,E2 -17120.514} C_VEL
LIN {X 0,Y 294.481,Z 345.329,A -85,B 0,C 180,E1 -17122.264,E2 -17122.264} C_VEL
LIN {X 0,Y 296.201,Z 332.079,A -85,B 0,C 180,E1 -17123.603,E2 -17123.603} C_VEL
LIN {X 0,Y 296.346,Z 330.266,A -85,B 0,C 180,E1 -17123.776,E2 -17123.776} C_VEL
LIN {X 0,Y 292.566,Z 314.741,A -85,B 0,C 180,E1 -17125.411,E2 -17125.411} C_VEL
LIN {X 0,Y 287.953,Z 298.31,A -85,B 0,C 180,E1 -17126.894,E2 -17126.894} C_VEL
LIN {X 0,Y 284.279,Z 287.073,A -85,B 0,C 180,E1 -17127.806,E2 -17127.806} C_VEL
LIN {X 0,Y 283.621,Z 284.782,A -85,B 0,C 180,E1 -17127.999,E2 -17127.999} C_VEL
LIN {X 0,Y 283.918,Z 284.746,A -85,B 0,C 180,E1 -17131.321,E2 -17131.321} C_VEL
LIN {X 0,Y 284.243,Z 284.705,A -85,B 0,C 180,E1 -17135.32,E2 -17135.32} C_VEL
LIN {X 0,Y 284.303,Z 284.695,A -85,B 0,C 180,E1 -17138.171,E2 -17138.171} C_VEL
LIN {X 0,Y 284.272,Z 284.699,A -85,B 0,C 180,E1 -17142.124,E2 -17142.124} C_VEL
LIN {X 0,Y 284.257,Z 284.7,A -85,B 0,C 180,E1 -17146.189,E2 -17146.189} C_VEL
LIN {X 0,Y 284.309,Z 284.693,A -85,B 0,C 180,E1 -17150.024,E2 -17150.024} C_VEL
LIN {X 0,Y 284.333,Z 284.69,A -85,B 0,C 180,E1 -17153.614,E2 -17153.614} C_VEL
LIN {X 0,Y 284.31,Z 284.694,A -85,B 0,C 180,E1 -17157.19,E2 -17157.19} C_VEL
LIN {X 0,Y 284.358,Z 284.689,A -85,B 0,C 180,E1 -17160.376,E2 -17160.376} C_VEL
LIN {X 0,Y 284.377,Z 284.684,A -85,B 0,C 180,E1 -17163.586,E2 -17163.586} C_VEL
LIN {X 0,Y 284.364,Z 284.688,A -85,B 0,C 180,E1 -17166.707,E2 -17166.707} C_VEL
LIN {X 0,Y 284.402,Z 284.681,A -85,B 0,C 180,E1 -17171.261,E2 -17171.261} C_VEL
LIN {X 0,Y 284.495,Z 284.672,A -85,B 0,C 180,E1 -17174.459,E2 -17174.459} C_VEL
LIN {X 0,Y 284.491,Z 284.672,A -85,B 0,C 180,E1 -17178.602,E2 -17178.602} C_VEL
LIN {X 0,Y 284.611,Z 284.655,A -85,B 0,C 180,E1 -17181.48,E2 -17181.48} C_VEL
LIN {X 0,Y 284.576,Z 284.662,A -85,B 0,C 180,E1 -17184.331,E2 -17184.331} C_VEL
LIN {X 0,Y 284.855,Z 284.625,A -85,B 0,C 180,E1 -17188.586,E2 -17188.586} C_VEL
LIN {X 0,Y 284.854,Z 284.625,A -85,B 0,C 180,E1 -17191.414,E2 -17191.414} C_VEL
LIN {X 0,Y 284.654,Z 284.65,A -85,B 0,C 180,E1 -17197.091,E2 -17197.091} C_VEL
LIN {X 0,Y 284.517,Z 284.669,A -85,B 0,C 180,E1 -17199.957,E2 -17199.957} C_VEL
LIN {X 0,Y 284.485,Z 284.671,A -85,B 0,C 180,E1 -17204.303,E2 -17204.303} C_VEL
LIN {X 0,Y 284.429,Z 284.679,A -85,B 0,C 180,E1 -17207.248,E2 -17207.248} C_VEL
LIN {X 0,Y 284.384,Z 284.684,A -85,B 0,C 180,E1 -17210.242,E2 -17210.242} C_VEL
LIN {X 0,Y 284.372,Z 284.686,A -85,B 0,C 180,E1 -17213.875,E2 -17213.875} C_VEL
LIN {X 0,Y 284.397,Z 284.684,A -85,B 0,C 180,E1 -17217.172,E2 -17217.172} C_VEL
LIN {X 0,Y 284.297,Z 284.699,A -85,B 0,C 180,E1 -17221.274,E2 -17221.274} C_VEL
LIN {X 0,Y 284.339,Z 284.692,A -85,B 0,C 180,E1 -17225.347,E2 -17225.347} C_VEL
LIN {X 0,Y 284.3,Z 284.694,A -85,B 0,C 180,E1 -17228.171,E2 -17228.171} C_VEL
LIN {X 0,Y 284.24,Z 284.7,A -85,B 0,C 180,E1 -17232.117,E2 -17232.117} C_VEL
LIN {X 0,Y 284.258,Z 284.699,A -85,B 0,C 180,E1 -17236.189,E2 -17236.189} C_VEL
LIN {X 0,Y 284.309,Z 284.692,A -85,B 0,C 180,E1 -17240.024,E2 -17240.024} C_VEL
LIN {X 0,Y 284.334,Z 284.69,A -85,B 0,C 180,E1 -17243.614,E2 -17243.614} C_VEL
LIN {X 0,Y 284.311,Z 284.693,A -85,B 0,C 180,E1 -17247.19,E2 -17247.19} C_VEL
LIN {X 0,Y 284.359,Z 284.688,A -85,B 0,C 180,E1 -17250.376,E2 -17250.376} C_VEL
LIN {X 0,Y 284.378,Z 284.684,A -85,B 0,C 180,E1 -17253.586,E2 -17253.586} C_VEL
LIN {X 0,Y 284.366,Z 284.688,A -85,B 0,C 180,E1 -17256.707,E2 -17256.707} C_VEL
LIN {X 0,Y 284.407,Z 284.681,A -85,B 0,C 180,E1 -17261.261,E2 -17261.261} C_VEL
LIN {X 0,Y 284.496,Z 284.672,A -85,B 0,C 180,E1 -17264.459,E2 -17264.459} C_VEL
LIN {X 0,Y 284.487,Z 284.673,A -85,B 0,C 180,E1 -17268.601,E2 -17268.601} C_VEL
LIN {X 0,Y 284.612,Z 284.655,A -85,B 0,C 180,E1 -17271.479,E2 -17271.479} C_VEL
LIN {X 0,Y 284.577,Z 284.662,A -85,B 0,C 180,E1 -17274.33,E2 -17274.33} C_VEL
LIN {X 0,Y 284.856,Z 284.625,A -85,B 0,C 180,E1 -17278.586,E2 -17278.586} C_VEL
LIN {X 0,Y 284.855,Z 284.625,A -85,B 0,C 180,E1 -17281.413,E2 -17281.413} C_VEL
LIN {X 0,Y 284.58,Z 284.662,A -85,B 0,C 180,E1 -17285.669,E2 -17285.669} C_VEL
LIN {X 0,Y 284.611,Z 284.654,A -85,B 0,C 180,E1 -17288.981,E2 -17288.981} C_VEL
LIN {X 0,Y 284.478,Z 284.671,A -85,B 0,C 180,E1 -17292.846,E2 -17292.846} C_VEL
LIN {X 0,Y 284.478,Z 284.672,A -85,B 0,C 180,E1 -17294.2,E2 -17294.2} C_VEL
LIN {X 0,Y 283.875,Z 284.753,A -85,B 0,C 180,E1 -17295.38,E2 -17295.38} C_VEL
LIN {X 0,Y 281.062,Z 285.105,A -85,B 0,C 180,E1 -17297.303,E2 -17297.303} C_VEL
LIN {X 0,Y 278.59,Z 285.409,A -85,B 0,C 180,E1 -17298.864,E2 -17298.864} C_VEL
LIN {X 0,Y 277.459,Z 285.548,A -85,B 0,C 180,E1 -17300.073,E2 -17300.073} C_VEL
LIN {X 0,Y 277.331,Z 285.562,A -85,B 0,C 180,E1 -17300.484,E2 -17300.484} C_VEL
LIN {X 0,Y 277.282,Z 285.57,A -85,B 0,C 180,E1 -17304.152,E2 -17304.152} C_VEL
LIN {X 0,Y 277.263,Z 285.66,A -85,B 0,C 180,E1 -17308.243,E2 -17308.243} C_VEL
LIN {X 0,Y 277.877,Z 289.514,A -85,B 0,C 180,E1 -17312.081,E2 -17312.081} C_VEL
LIN {X 0,Y 278.625,Z 293.895,A -85,B 0,C 180,E1 -17316.18,E2 -17316.18} C_VEL
LIN {X 0,Y 279.418,Z 298.094,A -85,B 0,C 180,E1 -17319.895,E2 -17319.895} C_VEL
LIN {X 0,Y 280.284,Z 302.186,A -85,B 0,C 180,E1 -17323.35,E2 -17323.35} C_VEL
LIN {X 0,Y 280.819,Z 306.159,A -85,B 0,C 180,E1 -17326.533,E2 -17326.533} C_VEL
LIN {X 0,Y 280.519,Z 309.92,A -85,B 0,C 180,E1 -17329.353,E2 -17329.353} C_VEL
LIN {X 0,Y 279.665,Z 314.827,A -85,B 0,C 180,E1 -17332.906,E2 -17332.906} C_VEL
LIN {X 0,Y 279.221,Z 317.093,A -85,B 0,C 180,E1 -17334.512,E2 -17334.512} C_VEL
LIN {X 0,Y 283.236,Z 335.185,A -85,B 0,C 180,E1 -17335.922,E2 -17335.922} C_VEL
LIN {X 0,Y 286.571,Z 351.314,A -85,B 0,C 180,E1 -17337.428,E2 -17337.428} C_VEL
LIN {X 0,Y 289.321,Z 366.078,A -85,B 0,C 180,E1 -17339.023,E2 -17339.023} C_VEL
LIN {X 0,Y 291.481,Z 380.353,A -85,B 0,C 180,E1 -17340.786,E2 -17340.786} C_VEL
LIN {X 0,Y 288.781,Z 393.922,A -85,B 0,C 180,E1 -17342.458,E2 -17342.458} C_VEL
LIN {X 0,Y 285.926,Z 407.572,A -85,B 0,C 180,E1 -17344.523,E2 -17344.523} C_VEL
LIN {X 0,Y 283.47,Z 419.089,A -85,B 0,C 180,E1 -17346.629,E2 -17346.629} C_VEL
LIN {X 0,Y 281.156,Z 430.395,A -85,B 0,C 180,E1 -17349.133,E2 -17349.133} C_VEL
LIN {X 0,Y 279.166,Z 439.842,A -85,B 0,C 180,E1 -17351.658,E2 -17351.658} C_VEL
LIN {X 0,Y 277.624,Z 448.135,A -85,B 0,C 180,E1 -17354.345,E2 -17354.345} C_VEL
LIN {X 0,Y 276.648,Z 454.368,A -85,B 0,C 180,E1 -17356.783,E2 -17356.783} C_VEL
LIN {X 0,Y 275.903,Z 460.398,A -85,B 0,C 180,E1 -17359.729,E2 -17359.729} C_VEL
LIN {X 0,Y 275.57,Z 464.981,A -85,B 0,C 180,E1 -17362.674,E2 -17362.674} C_VEL
LIN {X 0,Y 275.506,Z 468.202,A -85,B 0,C 180,E1 -17365.611,E2 -17365.611} C_VEL
LIN {X 0,Y 275.444,Z 470.128,A -85,B 0,C 180,E1 -17368.538,E2 -17368.538} C_VEL
LIN {X 0,Y 275.498,Z 470.634,A -85,B 0,C 180,E1 -17370,E2 -17370} C_VEL
LIN {X 0,Y 275.393,Z 470.724,A -85,B 0,C 180,E1 -17372.926,E2 -17372.926} C_VEL
LIN {X 0,Y 275.39,Z 469.635,A -85,B 0,C 180,E1 -17375.859,E2 -17375.859} C_VEL
LIN {X 0,Y 275.579,Z 467.342,A -85,B 0,C 180,E1 -17378.802,E2 -17378.802} C_VEL
LIN {X 0,Y 276.413,Z 462.952,A -85,B 0,C 180,E1 -17382.481,E2 -17382.481} C_VEL
LIN {X 0,Y 278.093,Z 456.773,A -85,B 0,C 180,E1 -17386.141,E2 -17386.141} C_VEL
LIN {X 0,Y 280.226,Z 450.515,A -85,B 0,C 180,E1 -17389.029,E2 -17389.029} C_VEL
LIN {X 0,Y 283.418,Z 442.031,A -85,B 0,C 180,E1 -17392.22,E2 -17392.22} C_VEL
LIN {X 0,Y 287.242,Z 432.603,A -85,B 0,C 180,E1 -17395.139,E2 -17395.139} C_VEL
LIN {X 0,Y 292.15,Z 421.435,A -85,B 0,C 180,E1 -17397.976,E2 -17397.976} C_VEL
LIN {X 0,Y 297.61,Z 409.358,A -85,B 0,C 180,E1 -17400.512,E2 -17400.512} C_VEL
LIN {X 0,Y 303.109,Z 397.413,A -85,B 0,C 180,E1 -17402.606,E2 -17402.606} C_VEL
LIN {X 0,Y 305.545,Z 391.788,A -85,B 0,C 180,E1 -17403.507,E2 -17403.507} C_VEL
LIN {X 0,Y 309.048,Z 379.533,A -85,B 0,C 180,E1 -17405.844,E2 -17405.844} C_VEL
LIN {X 0,Y 310.627,Z 371.604,A -85,B 0,C 180,E1 -17407.653,E2 -17407.653} C_VEL
LIN {X 0,Y 311.512,Z 365.41,A -85,B 0,C 180,E1 -17409.448,E2 -17409.448} C_VEL
LIN {X 0,Y 312.075,Z 361.694,A -85,B 0,C 180,E1 -17410.775,E2 -17410.775} C_VEL
LIN {X 0,Y 312.721,Z 358.213,A -85,B 0,C 180,E1 -17412.393,E2 -17412.393} C_VEL
LIN {X 0,Y 313.359,Z 355.867,A -85,B 0,C 180,E1 -17414.136,E2 -17414.136} C_VEL
LIN {X 0,Y 314.029,Z 355.144,A -85,B 0,C 180,E1 -17416.07,E2 -17416.07} C_VEL
LIN {X 0,Y 314.712,Z 356.099,A -85,B 0,C 180,E1 -17417.937,E2 -17417.937} C_VEL
LIN {X 0,Y 315.486,Z 358.384,A -85,B 0,C 180,E1 -17419.758,E2 -17419.758} C_VEL
LIN {X 0,Y 315.929,Z 361.165,A -85,B 0,C 180,E1 -17421.132,E2 -17421.132} C_VEL
LIN {X 0,Y 315.934,Z 362.818,A -85,B 0,C 180,E1 -17421.725,E2 -17421.725} C_VEL
LIN {X 0,Y 309.373,Z 376.758,A -85,B 0,C 180,E1 -17423.798,E2 -17423.798} C_VEL
LIN {X 0,Y 303.795,Z 388.186,A -85,B 0,C 180,E1 -17425.875,E2 -17425.875} C_VEL
LIN {X 0,Y 298.147,Z 399.392,A -85,B 0,C 180,E1 -17428.344,E2 -17428.344} C_VEL
LIN {X 0,Y 293.739,Z 408.007,A -85,B 0,C 180,E1 -17430.628,E2 -17430.628} C_VEL
LIN {X 0,Y 289.396,Z 416.329,A -85,B 0,C 180,E1 -17433.303,E2 -17433.303} C_VEL
LIN {X 0,Y 285.705,Z 423.253,A -85,B 0,C 180,E1 -17436.054,E2 -17436.054} C_VEL
LIN {X 0,Y 282.7,Z 428.843,A -85,B 0,C 180,E1 -17438.871,E2 -17438.871} C_VEL
LIN {X 0,Y 280.866,Z 432.222,A -85,B 0,C 180,E1 -17441.017,E2 -17441.017} C_VEL
LIN {X 0,Y 278.964,Z 435.622,A -85,B 0,C 180,E1 -17443.912,E2 -17443.912} C_VEL
LIN {X 0,Y 277.438,Z 437.843,A -85,B 0,C 180,E1 -17446.822,E2 -17446.822} C_VEL
LIN {X 0,Y 276.495,Z 438.901,A -85,B 0,C 180,E1 -17449.751,E2 -17449.751} C_VEL
LIN {X 0,Y 275.92,Z 438.776,A -85,B 0,C 180,E1 -17452.684,E2 -17452.684} C_VEL
LIN {X 0,Y 275.698,Z 437.454,A -85,B 0,C 180,E1 -17455.614,E2 -17455.614} C_VEL
LIN {X 0,Y 275.595,Z 434.926,A -85,B 0,C 180,E1 -17458.539,E2 -17458.539} C_VEL
LIN {X 0,Y 275.656,Z 431.11,A -85,B 0,C 180,E1 -17461.461,E2 -17461.461} C_VEL
LIN {X 0,Y 276.136,Z 425.934,A -85,B 0,C 180,E1 -17464.379,E2 -17464.379} C_VEL
LIN {X 0,Y 276.705,Z 421.085,A -85,B 0,C 180,E1 -17466.563,E2 -17466.563} C_VEL
LIN {X 0,Y 277.473,Z 413.267,A -85,B 0,C 180,E1 -17469.476,E2 -17469.476} C_VEL
LIN {X 0,Y 278.638,Z 404.964,A -85,B 0,C 180,E1 -17472.011,E2 -17472.011} C_VEL
LIN {X 0,Y 280.175,Z 395.042,A -85,B 0,C 180,E1 -17474.528,E2 -17474.528} C_VEL
LIN {X 0,Y 281.992,Z 383.216,A -85,B 0,C 180,E1 -17477.029,E2 -17477.029} C_VEL
LIN {X 0,Y 284.079,Z 370.121,A -85,B 0,C 180,E1 -17479.323,E2 -17479.323} C_VEL
LIN {X 0,Y 285.874,Z 357.723,A -85,B 0,C 180,E1 -17481.14,E2 -17481.14} C_VEL
LIN {X 0,Y 287.86,Z 344.134,A -85,B 0,C 180,E1 -17482.805,E2 -17482.805} C_VEL
LIN {X 0,Y 289.411,Z 332.439,A -85,B 0,C 180,E1 -17484.002,E2 -17484.002} C_VEL
LIN {X 0,Y 288.797,Z 328.522,A -85,B 0,C 180,E1 -17484.438,E2 -17484.438} C_VEL
LIN {X 0,Y 285.281,Z 314.297,A -85,B 0,C 180,E1 -17485.949,E2 -17485.949} C_VEL
LIN {X 0,Y 280.703,Z 298.026,A -85,B 0,C 180,E1 -17487.461,E2 -17487.461} C_VEL
LIN {X 0,Y 276.616,Z 285.655,A -85,B 0,C 180,E1 -17488.554,E2 -17488.554} C_VEL
LIN {X 0,Y 277.046,Z 285.602,A -85,B 0,C 180,E1 -17493.161,E2 -17493.161} C_VEL
LIN {X 0,Y 277.217,Z 285.578,A -85,B 0,C 180,E1 -17495.78,E2 -17495.78} C_VEL
LIN {X 0,Y 277.233,Z 285.579,A -85,B 0,C 180,E1 -17499.329,E2 -17499.329} C_VEL
LIN {X 0,Y 277.212,Z 285.581,A -85,B 0,C 180,E1 -17503.198,E2 -17503.198} C_VEL
LIN {X 0,Y 277.217,Z 285.577,A -85,B 0,C 180,E1 -17507.325,E2 -17507.325} C_VEL
LIN {X 0,Y 277.264,Z 285.57,A -85,B 0,C 180,E1 -17511.793,E2 -17511.793} C_VEL
LIN {X 0,Y 277.287,Z 285.569,A -85,B 0,C 180,E1 -17514.342,E2 -17514.342} C_VEL
LIN {X 0,Y 277.247,Z 285.573,A -85,B 0,C 180,E1 -17517.836,E2 -17517.836} C_VEL
LIN {X 0,Y 277.27,Z 285.57,A -85,B 0,C 180,E1 -17521.21,E2 -17521.21} C_VEL
LIN {X 0,Y 277.314,Z 285.569,A -85,B 0,C 180,E1 -17524.479,E2 -17524.479} C_VEL
LIN {X 0,Y 277.28,Z 285.568,A -85,B 0,C 180,E1 -17527.654,E2 -17527.654} C_VEL
LIN {X 0,Y 277.345,Z 285.562,A -85,B 0,C 180,E1 -17530.766,E2 -17530.766} C_VEL
LIN {X 0,Y 277.438,Z 285.547,A -85,B 0,C 180,E1 -17535.326,E2 -17535.326} C_VEL
LIN {X 0,Y 277.463,Z 285.547,A -85,B 0,C 180,E1 -17539.787,E2 -17539.787} C_VEL
LIN {X 0,Y 277.604,Z 285.527,A -85,B 0,C 180,E1 -17542.728,E2 -17542.728} C_VEL
LIN {X 0,Y 277.821,Z 285.502,A -85,B 0,C 180,E1 -17548.55,E2 -17548.55} C_VEL
LIN {X 0,Y 277.821,Z 285.501,A -85,B 0,C 180,E1 -17551.45,E2 -17551.45} C_VEL
LIN {X 0,Y 277.612,Z 285.528,A -85,B 0,C 180,E1 -17557.272,E2 -17557.272} C_VEL
LIN {X 0,Y 277.46,Z 285.546,A -85,B 0,C 180,E1 -17560.213,E2 -17560.213} C_VEL
LIN {X 0,Y 277.438,Z 285.548,A -85,B 0,C 180,E1 -17564.674,E2 -17564.674} C_VEL
LIN {X 0,Y 277.348,Z 285.561,A -85,B 0,C 180,E1 -17569.234,E2 -17569.234} C_VEL
LIN {X 0,Y 277.332,Z 285.563,A -85,B 0,C 180,E1 -17573.92,E2 -17573.92} C_VEL
LIN {X 0,Y 277.326,Z 285.566,A -85,B 0,C 180,E1 -17577.504,E2 -17577.504} C_VEL
LIN {X 0,Y 277.275,Z 285.569,A -85,B 0,C 180,E1 -17580.481,E2 -17580.481} C_VEL
LIN {X 0,Y 277.249,Z 285.571,A -85,B 0,C 180,E1 -17583.896,E2 -17583.896} C_VEL
LIN {X 0,Y 277.258,Z 285.573,A -85,B 0,C 180,E1 -17587.471,E2 -17587.471} C_VEL
LIN {X 0,Y 277.187,Z 285.582,A -85,B 0,C 180,E1 -17591.241,E2 -17591.241} C_VEL
LIN {X 0,Y 277.2,Z 285.581,A -85,B 0,C 180,E1 -17595.227,E2 -17595.227} C_VEL
LIN {X 0,Y 277.226,Z 285.575,A -85,B 0,C 180,E1 -17599.512,E2 -17599.512} C_VEL
LIN {X 0,Y 277.268,Z 285.571,A -85,B 0,C 180,E1 -17602.53,E2 -17602.53} C_VEL
LIN {X 0,Y 277.25,Z 285.573,A -85,B 0,C 180,E1 -17606.104,E2 -17606.104} C_VEL
LIN {X 0,Y 277.265,Z 285.569,A -85,B 0,C 180,E1 -17609.539,E2 -17609.539} C_VEL
LIN {X 0,Y 277.359,Z 285.561,A -85,B 0,C 180,E1 -17612.864,E2 -17612.864} C_VEL
LIN {X 0,Y 277.33,Z 285.563,A -85,B 0,C 180,E1 -17616.079,E2 -17616.079} C_VEL
LIN {X 0,Y 277.348,Z 285.562,A -85,B 0,C 180,E1 -17620.766,E2 -17620.766} C_VEL
LIN {X 0,Y 277.439,Z 285.547,A -85,B 0,C 180,E1 -17625.326,E2 -17625.326} C_VEL
LIN {X 0,Y 277.461,Z 285.547,A -85,B 0,C 180,E1 -17629.787,E2 -17629.787} C_VEL
LIN {X 0,Y 277.605,Z 285.528,A -85,B 0,C 180,E1 -17632.727,E2 -17632.727} C_VEL
LIN {X 0,Y 277.822,Z 285.502,A -85,B 0,C 180,E1 -17638.55,E2 -17638.55} C_VEL
LIN {X 0,Y 277.821,Z 285.501,A -85,B 0,C 180,E1 -17641.449,E2 -17641.449} C_VEL
LIN {X 0,Y 277.55,Z 285.539,A -85,B 0,C 180,E1 -17645.813,E2 -17645.813} C_VEL
LIN {X 0,Y 277.563,Z 285.533,A -85,B 0,C 180,E1 -17649.068,E2 -17649.068} C_VEL
LIN {X 0,Y 277.419,Z 285.552,A -85,B 0,C 180,E1 -17653.179,E2 -17653.179} C_VEL
LIN {X 0,Y 277.409,Z 285.553,A -85,B 0,C 180,E1 -17656.181,E2 -17656.181} C_VEL
LIN {X 0,Y 277.331,Z 285.562,A -85,B 0,C 180,E1 -17660.484,E2 -17660.484} C_VEL
LIN {X 0,Y 276.556,Z 285.663,A -85,B 0,C 180,E1 -17661.696,E2 -17661.696} C_VEL
LIN {X 0,Y 273.637,Z 286.026,A -85,B 0,C 180,E1 -17663.671,E2 -17663.671} C_VEL
LIN {X 0,Y 271.255,Z 286.323,A -85,B 0,C 180,E1 -17665.275,E2 -17665.275} C_VEL
LIN {X 0,Y 270.286,Z 286.443,A -85,B 0,C 180,E1 -17666.519,E2 -17666.519} C_VEL
LIN {X 0,Y 270.232,Z 286.449,A -85,B 0,C 180,E1 -17666.94,E2 -17666.94} C_VEL
LIN {X 0,Y 270.252,Z 286.597,A -85,B 0,C 180,E1 -17667.91,E2 -17667.91} C_VEL
LIN {X 0,Y 270.766,Z 289.899,A -85,B 0,C 180,E1 -17671.273,E2 -17671.273} C_VEL
LIN {X 0,Y 271.324,Z 293.487,A -85,B 0,C 180,E1 -17674.74,E2 -17674.74} C_VEL
LIN {X 0,Y 272.252,Z 298.402,A -85,B 0,C 180,E1 -17679.246,E2 -17679.246} C_VEL
LIN {X 0,Y 273.166,Z 302.706,A -85,B 0,C 180,E1 -17682.983,E2 -17682.983} C_VEL
LIN {X 0,Y 273.709,Z 306.502,A -85,B 0,C 180,E1 -17686.109,E2 -17686.109} C_VEL
LIN {X 0,Y 273.687,Z 309.088,A -85,B 0,C 180,E1 -17688.132,E2 -17688.132} C_VEL
LIN {X 0,Y 272.826,Z 314.005,A -85,B 0,C 180,E1 -17691.812,E2 -17691.812} C_VEL
LIN {X 0,Y 272.308,Z 316.839,A -85,B 0,C 180,E1 -17693.842,E2 -17693.842} C_VEL
LIN {X 0,Y 276.309,Z 335.109,A -85,B 0,C 180,E1 -17695.32,E2 -17695.32} C_VEL
LIN {X 0,Y 279.762,Z 352.217,A -85,B 0,C 180,E1 -17696.974,E2 -17696.974} C_VEL
LIN {X 0,Y 282.552,Z 367.597,A -85,B 0,C 180,E1 -17698.718,E2 -17698.718} C_VEL
LIN {X 0,Y 284.509,Z 380.677,A -85,B 0,C 180,E1 -17700.393,E2 -17700.393} C_VEL
LIN {X 0,Y 283.316,Z 387.782,A -85,B 0,C 180,E1 -17701.274,E2 -17701.274} C_VEL
LIN {X 0,Y 280.41,Z 401.242,A -85,B 0,C 180,E1 -17703.183,E2 -17703.183} C_VEL
LIN {X 0,Y 277.727,Z 413.635,A -85,B 0,C 180,E1 -17705.321,E2 -17705.321} C_VEL
LIN {X 0,Y 275.382,Z 424.159,A -85,B 0,C 180,E1 -17707.492,E2 -17707.492} C_VEL
LIN {X 0,Y 273.158,Z 434.546,A -85,B 0,C 180,E1 -17710.068,E2 -17710.068} C_VEL
LIN {X 0,Y 271.408,Z 443.263,A -85,B 0,C 180,E1 -17712.675,E2 -17712.675} C_VEL
LIN {X 0,Y 269.935,Z 451.44,A -85,B 0,C 180,E1 -17715.68,E2 -17715.68} C_VEL
LIN {X 0,Y 269.024,Z 457.988,A -85,B 0,C 180,E1 -17718.701,E2 -17718.701} C_VEL
LIN {X 0,Y 268.597,Z 463.067,A -85,B 0,C 180,E1 -17721.726,E2 -17721.726} C_VEL
LIN {X 0,Y 268.471,Z 466.107,A -85,B 0,C 180,E1 -17724.13,E2 -17724.13} C_VEL
LIN {X 0,Y 268.34,Z 468.627,A -85,B 0,C 180,E1 -17726.997,E2 -17726.997} C_VEL
LIN {X 0,Y 268.419,Z 470.067,A -85,B 0,C 180,E1 -17730,E2 -17730} C_VEL
LIN {X 0,Y 268.321,Z 470.281,A -85,B 0,C 180,E1 -17733.003,E2 -17733.003} C_VEL
LIN {X 0,Y 268.302,Z 469.259,A -85,B 0,C 180,E1 -17736.014,E2 -17736.014} C_VEL
LIN {X 0,Y 268.504,Z 467.109,A -85,B 0,C 180,E1 -17739.036,E2 -17739.036} C_VEL
LIN {X 0,Y 269.13,Z 463.882,A -85,B 0,C 180,E1 -17742.059,E2 -17742.059} C_VEL
LIN {X 0,Y 270.391,Z 459.562,A -85,B 0,C 180,E1 -17745.065,E2 -17745.065} C_VEL
LIN {X 0,Y 272.852,Z 452.547,A -85,B 0,C 180,E1 -17748.782,E2 -17748.782} C_VEL
LIN {X 0,Y 275.645,Z 445.662,A -85,B 0,C 180,E1 -17751.697,E2 -17751.697} C_VEL
LIN {X 0,Y 279.611,Z 436.505,A -85,B 0,C 180,E1 -17754.892,E2 -17754.892} C_VEL
LIN {X 0,Y 284.735,Z 425.646,A -85,B 0,C 180,E1 -17757.968,E2 -17757.968} C_VEL
LIN {X 0,Y 290.221,Z 414.534,A -85,B 0,C 180,E1 -17760.567,E2 -17760.567} C_VEL
LIN {X 0,Y 296.589,Z 401.809,A -85,B 0,C 180,E1 -17763.026,E2 -17763.026} C_VEL
LIN {X 0,Y 300.097,Z 394.773,A -85,B 0,C 180,E1 -17764.198,E2 -17764.198} C_VEL
LIN {X 0,Y 304.137,Z 383.216,A -85,B 0,C 180,E1 -17766.515,E2 -17766.515} C_VEL
LIN {X 0,Y 306.085,Z 375.755,A -85,B 0,C 180,E1 -17768.312,E2 -17768.312} C_VEL
LIN {X 0,Y 307.38,Z 369.628,A -85,B 0,C 180,E1 -17770.206,E2 -17770.206} C_VEL
LIN {X 0,Y 308.52,Z 364.861,A -85,B 0,C 180,E1 -17772.166,E2 -17772.166} C_VEL
LIN {X 0,Y 309.044,Z 362.977,A -85,B 0,C 180,E1 -17773.305,E2 -17773.305} C_VEL
LIN {X 0,Y 309.634,Z 361.542,A -85,B 0,C 180,E1 -17774.719,E2 -17774.719} C_VEL
LIN {X 0,Y 310.239,Z 361.235,A -85,B 0,C 180,E1 -17776.462,E2 -17776.462} C_VEL
LIN {X 0,Y 310.815,Z 362.358,A -85,B 0,C 180,E1 -17778.261,E2 -17778.261} C_VEL
LIN {X 0,Y 311.099,Z 363.252,A -85,B 0,C 180,E1 -17779.07,E2 -17779.07} C_VEL
LIN {X 0,Y 311.379,Z 364.941,A -85,B 0,C 180,E1 -17780.121,E2 -17780.121} C_VEL
LIN {X 0,Y 311.459,Z 366.406,A -85,B 0,C 180,E1 -17780.816,E2 -17780.816} C_VEL
LIN {X 0,Y 309.517,Z 370.457,A -85,B 0,C 180,E1 -17781.482,E2 -17781.482} C_VEL
LIN {X 0,Y 303.388,Z 382.079,A -85,B 0,C 180,E1 -17783.381,E2 -17783.381} C_VEL
LIN {X 0,Y 296.613,Z 394.598,A -85,B 0,C 180,E1 -17785.898,E2 -17785.898} C_VEL
LIN {X 0,Y 290.39,Z 405.668,A -85,B 0,C 180,E1 -17788.645,E2 -17788.645} C_VEL
LIN {X 0,Y 285.472,Z 414.328,A -85,B 0,C 180,E1 -17791.311,E2 -17791.311} C_VEL
LIN {X 0,Y 281.137,Z 421.812,A -85,B 0,C 180,E1 -17794.152,E2 -17794.152} C_VEL
LIN {X 0,Y 277.679,Z 427.596,A -85,B 0,C 180,E1 -17796.903,E2 -17796.903} C_VEL
LIN {X 0,Y 274.827,Z 432.313,A -85,B 0,C 180,E1 -17799.805,E2 -17799.805} C_VEL
LIN {X 0,Y 272.786,Z 435.523,A -85,B 0,C 180,E1 -17802.414,E2 -17802.414} C_VEL
LIN {X 0,Y 271.23,Z 437.756,A -85,B 0,C 180,E1 -17804.983,E2 -17804.983} C_VEL
LIN {X 0,Y 269.943,Z 439.231,A -85,B 0,C 180,E1 -17807.979,E2 -17807.979} C_VEL
LIN {X 0,Y 269.14,Z 439.556,A -85,B 0,C 180,E1 -17810.986,E2 -17810.986} C_VEL
LIN {X 0,Y 268.717,Z 438.701,A -85,B 0,C 180,E1 -17813.995,E2 -17813.995} C_VEL
LIN {X 0,Y 268.545,Z 436.658,A -85,B 0,C 180,E1 -17817,E2 -17817} C_VEL
LIN {X 0,Y 268.503,Z 433.375,A -85,B 0,C 180,E1 -17820,E2 -17820} C_VEL
LIN {X 0,Y 268.763,Z 428.794,A -85,B 0,C 180,E1 -17822.998,E2 -17822.998} C_VEL
LIN {X 0,Y 269.477,Z 422.796,A -85,B 0,C 180,E1 -17825.988,E2 -17825.988} C_VEL
LIN {X 0,Y 270.187,Z 415.229,A -85,B 0,C 180,E1 -17828.979,E2 -17828.979} C_VEL
LIN {X 0,Y 271.273,Z 407.205,A -85,B 0,C 180,E1 -17831.583,E2 -17831.583} C_VEL
LIN {X 0,Y 272.802,Z 397.649,A -85,B 0,C 180,E1 -17834.167,E2 -17834.167} C_VEL
LIN {X 0,Y 274.561,Z 386.253,A -85,B 0,C 180,E1 -17836.737,E2 -17836.737} C_VEL
LIN {X 0,Y 276.451,Z 374.695,A -85,B 0,C 180,E1 -17838.914,E2 -17838.914} C_VEL
LIN {X 0,Y 278.489,Z 361.635,A -85,B 0,C 180,E1 -17840.974,E2 -17840.974} C_VEL
LIN {X 0,Y 280.63,Z 347.362,A -85,B 0,C 180,E1 -17842.841,E2 -17842.841} C_VEL
LIN {X 0,Y 282.429,Z 334.463,A -85,B 0,C 180,E1 -17844.242,E2 -17844.242} C_VEL
LIN {X 0,Y 282.557,Z 332.66,A -85,B 0,C 180,E1 -17844.426,E2 -17844.426} C_VEL
LIN {X 0,Y 278.965,Z 317.535,A -85,B 0,C 180,E1 -17846.133,E2 -17846.133} C_VEL
LIN {X 0,Y 274.769,Z 302.074,A -85,B 0,C 180,E1 -17847.671,E2 -17847.671} C_VEL
LIN {X 0,Y 270.415,Z 289.029,A -85,B 0,C 180,E1 -17848.829,E2 -17848.829} C_VEL
LIN {X 0,Y 269.632,Z 286.524,A -85,B 0,C 180,E1 -17849.052,E2 -17849.052} C_VEL
LIN {X 0,Y 270.025,Z 286.474,A -85,B 0,C 180,E1 -17853.605,E2 -17853.605} C_VEL
LIN {X 0,Y 270.189,Z 286.455,A -85,B 0,C 180,E1 -17856.746,E2 -17856.746} C_VEL
LIN {X 0,Y 270.177,Z 286.457,A -85,B 0,C 180,E1 -17860.566,E2 -17860.566} C_VEL
LIN {X 0,Y 270.155,Z 286.459,A -85,B 0,C 180,E1 -17864.62,E2 -17864.62} C_VEL
LIN {X 0,Y 270.172,Z 286.458,A -85,B 0,C 180,E1 -17868.972,E2 -17868.972} C_VEL
LIN {X 0,Y 270.219,Z 286.449,A -85,B 0,C 180,E1 -17873.259,E2 -17873.259} C_VEL
LIN {X 0,Y 270.205,Z 286.453,A -85,B 0,C 180,E1 -17876.893,E2 -17876.893} C_VEL
LIN {X 0,Y 270.198,Z 286.453,A -85,B 0,C 180,E1 -17880.383,E2 -17880.383} C_VEL
LIN {X 0,Y 270.264,Z 286.442,A -85,B 0,C 180,E1 -17883.764,E2 -17883.764} C_VEL
LIN {X 0,Y 270.229,Z 286.446,A -85,B 0,C 180,E1 -17887.038,E2 -17887.038} C_VEL
LIN {X 0,Y 270.303,Z 286.441,A -85,B 0,C 180,E1 -17890.244,E2 -17890.244} C_VEL
LIN {X 0,Y 270.406,Z 286.424,A -85,B 0,C 180,E1 -17894.935,E2 -17894.935} C_VEL
LIN {X 0,Y 270.415,Z 286.424,A -85,B 0,C 180,E1 -17899.518,E2 -17899.518} C_VEL
LIN {X 0,Y 270.565,Z 286.405,A -85,B 0,C 180,E1 -17902.538,E2 -17902.538} C_VEL
LIN {X 0,Y 270.786,Z 286.378,A -85,B 0,C 180,E1 -17908.513,E2 -17908.513} C_VEL
LIN {X 0,Y 270.787,Z 286.377,A -85,B 0,C 180,E1 -17911.487,E2 -17911.487} C_VEL
LIN {X 0,Y 270.572,Z 286.406,A -85,B 0,C 180,E1 -17917.462,E2 -17917.462} C_VEL
LIN {X 0,Y 270.413,Z 286.423,A -85,B 0,C 180,E1 -17920.482,E2 -17920.482} C_VEL
LIN {X 0,Y 270.406,Z 286.425,A -85,B 0,C 180,E1 -17925.065,E2 -17925.065} C_VEL
LIN {X 0,Y 270.305,Z 286.44,A -85,B 0,C 180,E1 -17929.755,E2 -17929.755} C_VEL
LIN {X 0,Y 270.277,Z 286.44,A -85,B 0,C 180,E1 -17934.586,E2 -17934.586} C_VEL
LIN {X 0,Y 270.273,Z 286.442,A -85,B 0,C 180,E1 -17937.909,E2 -17937.909} C_VEL
LIN {X 0,Y 270.187,Z 286.456,A -85,B 0,C 180,E1 -17941.348,E2 -17941.348} C_VEL
LIN {X 0,Y 270.201,Z 286.451,A -85,B 0,C 180,E1 -17944.906,E2 -17944.906} C_VEL
LIN {X 0,Y 270.2,Z 286.452,A -85,B 0,C 180,E1 -17948.71,E2 -17948.71} C_VEL
LIN {X 0,Y 270.151,Z 286.459,A -85,B 0,C 180,E1 -17953.245,E2 -17953.245} C_VEL
LIN {X 0,Y 270.175,Z 286.454,A -85,B 0,C 180,E1 -17957.442,E2 -17957.442} C_VEL
LIN {X 0,Y 270.21,Z 286.449,A -85,B 0,C 180,E1 -17961.374,E2 -17961.374} C_VEL
LIN {X 0,Y 270.205,Z 286.452,A -85,B 0,C 180,E1 -17965.094,E2 -17965.094} C_VEL
LIN {X 0,Y 270.204,Z 286.45,A -85,B 0,C 180,E1 -17969.13,E2 -17969.13} C_VEL
LIN {X 0,Y 270.266,Z 286.443,A -85,B 0,C 180,E1 -17972.146,E2 -17972.146} C_VEL
LIN {X 0,Y 270.28,Z 286.44,A -85,B 0,C 180,E1 -17975.519,E2 -17975.519} C_VEL
LIN {X 0,Y 270.305,Z 286.44,A -85,B 0,C 180,E1 -17980.244,E2 -17980.244} C_VEL
LIN {X 0,Y 270.407,Z 286.424,A -85,B 0,C 180,E1 -17984.935,E2 -17984.935} C_VEL
LIN {X 0,Y 270.414,Z 286.424,A -85,B 0,C 180,E1 -17989.517,E2 -17989.517} C_VEL
LIN {X 0,Y 270.566,Z 286.405,A -85,B 0,C 180,E1 -17992.537,E2 -17992.537} C_VEL
LIN {X 0,Y 270.788,Z 286.378,A -85,B 0,C 180,E1 -17998.512,E2 -17998.512} C_VEL
LIN {X 0,Y 270.787,Z 286.377,A -85,B 0,C 180,E1 -18001.487,E2 -18001.487} C_VEL
LIN {X 0,Y 270.566,Z 286.406,A -85,B 0,C 180,E1 -18007.462,E2 -18007.462} C_VEL
LIN {X 0,Y 270.413,Z 286.423,A -85,B 0,C 180,E1 -18010.482,E2 -18010.482} C_VEL
LIN {X 0,Y 270.406,Z 286.425,A -85,B 0,C 180,E1 -18015.064,E2 -18015.064} C_VEL
LIN {X 0,Y 270.305,Z 286.441,A -85,B 0,C 180,E1 -18019.755,E2 -18019.755} C_VEL
LIN {X 0,Y 270.227,Z 286.448,A -85,B 0,C 180,E1 -18024.59,E2 -18024.59} C_VEL
LIN {X 0,Y 270.232,Z 286.449,A -85,B 0,C 180,E1 -18026.94,E2 -18026.94} C_VEL
LIN {X 0,Y 269.983,Z 286.735,A -85,B 0,C 180,E1 -18027.771,E2 -18027.771} C_VEL
LIN {X 0,Y 269.261,Z 287.442,A -85,B 0,C 180,E1 -18028.584,E2 -18028.584} C_VEL
LIN {X 0,Y 264.893,Z 291.439,A -85,B 0,C 180,E1 -18031.774,E2 -18031.774} C_VEL
LIN {X 0,Y 264.074,Z 292.838,A -85,B 0,C 180,E1 -18033.018,E2 -18033.018} C_VEL
LIN {X 0,Y 264.071,Z 293.274,A -85,B 0,C 180,E1 -18033.439,E2 -18033.439} C_VEL
LIN {X 0,Y 264.855,Z 297.645,A -85,B 0,C 180,E1 -18037.612,E2 -18037.612} C_VEL
LIN {X 0,Y 265.726,Z 301.816,A -85,B 0,C 180,E1 -18041.392,E2 -18041.392} C_VEL
LIN {X 0,Y 266.422,Z 305.514,A -85,B 0,C 180,E1 -18044.582,E2 -18044.582} C_VEL
LIN {X 0,Y 266.669,Z 309.143,A -85,B 0,C 180,E1 -18047.555,E2 -18047.555} C_VEL
LIN {X 0,Y 266.029,Z 313.138,A -85,B 0,C 180,E1 -18050.651,E2 -18050.651} C_VEL
LIN {X 0,Y 265.425,Z 316.592,A -85,B 0,C 180,E1 -18053.165,E2 -18053.165} C_VEL
LIN {X 0,Y 269.209,Z 334.262,A -85,B 0,C 180,E1 -18054.633,E2 -18054.633} C_VEL
LIN {X 0,Y 272.423,Z 350.126,A -85,B 0,C 180,E1 -18056.198,E2 -18056.198} C_VEL
LIN {X 0,Y 275.29,Z 366.378,A -85,B 0,C 180,E1 -18058.065,E2 -18058.065} C_VEL
LIN {X 0,Y 277.526,Z 380.952,A -85,B 0,C 180,E1 -18059.99,E2 -18059.99} C_VEL
LIN {X 0,Y 277.289,Z 383.922,A -85,B 0,C 180,E1 -18060.38,E2 -18060.38} C_VEL
LIN {X 0,Y 274.218,Z 397.917,A -85,B 0,C 180,E1 -18062.32,E2 -18062.32} C_VEL
LIN {X 0,Y 271.61,Z 409.738,A -85,B 0,C 180,E1 -18064.315,E2 -18064.315} C_VEL
LIN {X 0,Y 268.994,Z 421.041,A -85,B 0,C 180,E1 -18066.596,E2 -18066.596} C_VEL
LIN {X 0,Y 266.708,Z 431.594,A -85,B 0,C 180,E1 -18069.161,E2 -18069.161} C_VEL
LIN {X 0,Y 264.774,Z 440.687,A -85,B 0,C 180,E1 -18071.827,E2 -18071.827} C_VEL
LIN {X 0,Y 263.339,Z 448.297,A -85,B 0,C 180,E1 -18074.521,E2 -18074.521} C_VEL
LIN {X 0,Y 262.202,Z 455.385,A -85,B 0,C 180,E1 -18077.618,E2 -18077.618} C_VEL
LIN {X 0,Y 261.633,Z 460.949,A -85,B 0,C 180,E1 -18080.725,E2 -18080.725} C_VEL
LIN {X 0,Y 261.392,Z 465.103,A -85,B 0,C 180,E1 -18083.826,E2 -18083.826} C_VEL
LIN {X 0,Y 261.395,Z 466.683,A -85,B 0,C 180,E1 -18085.373,E2 -18085.373} C_VEL
LIN {X 0,Y 261.288,Z 468.857,A -85,B 0,C 180,E1 -18088.459,E2 -18088.459} C_VEL
LIN {X 0,Y 261.341,Z 469.488,A -85,B 0,C 180,E1 -18090,E2 -18090} C_VEL
LIN {X 0,Y 261.249,Z 469.777,A -85,B 0,C 180,E1 -18093.084,E2 -18093.084} C_VEL
LIN {X 0,Y 261.224,Z 468.886,A -85,B 0,C 180,E1 -18096.178,E2 -18096.178} C_VEL
LIN {X 0,Y 261.449,Z 466.897,A -85,B 0,C 180,E1 -18099.282,E2 -18099.282} C_VEL
LIN {X 0,Y 262.141,Z 463.836,A -85,B 0,C 180,E1 -18102.385,E2 -18102.385} C_VEL
LIN {X 0,Y 263.495,Z 459.645,A -85,B 0,C 180,E1 -18105.469,E2 -18105.469} C_VEL
LIN {X 0,Y 265.496,Z 454.4,A -85,B 0,C 180,E1 -18108.521,E2 -18108.521} C_VEL
LIN {X 0,Y 268.244,Z 448.078,A -85,B 0,C 180,E1 -18111.519,E2 -18111.519} C_VEL
LIN {X 0,Y 272.241,Z 439.588,A -85,B 0,C 180,E1 -18114.803,E2 -18114.803} C_VEL
LIN {X 0,Y 277.393,Z 429.583,A -85,B 0,C 180,E1 -18117.951,E2 -18117.951} C_VEL
LIN {X 0,Y 282.853,Z 419.351,A -85,B 0,C 180,E1 -18120.621,E2 -18120.621} C_VEL
LIN {X 0,Y 290.091,Z 406.088,A -85,B 0,C 180,E1 -18123.447,E2 -18123.447} C_VEL
LIN {X 0,Y 295.467,Z 396.21,A -85,B 0,C 180,E1 -18125.227,E2 -18125.227} C_VEL
LIN {X 0,Y 299.193,Z 386.899,A -85,B 0,C 180,E1 -18127.198,E2 -18127.198} C_VEL
LIN {X 0,Y 301.544,Z 379.816,A -85,B 0,C 180,E1 -18128.997,E2 -18128.997} C_VEL
LIN {X 0,Y 302.893,Z 375.111,A -85,B 0,C 180,E1 -18130.518,E2 -18130.518} C_VEL
LIN {X 0,Y 304.242,Z 370.739,A -85,B 0,C 180,E1 -18132.337,E2 -18132.337} C_VEL
LIN {X 0,Y 305.074,Z 368.475,A -85,B 0,C 180,E1 -18133.719,E2 -18133.719} C_VEL
LIN {X 0,Y 305.852,Z 367.089,A -85,B 0,C 180,E1 -18135.425,E2 -18135.425} C_VEL
LIN {X 0,Y 306.186,Z 367.067,A -85,B 0,C 180,E1 -18136.481,E2 -18136.481} C_VEL
LIN {X 0,Y 306.671,Z 368.254,A -85,B 0,C 180,E1 -18138.349,E2 -18138.349} C_VEL
LIN {X 0,Y 306.808,Z 369.145,A -85,B 0,C 180,E1 -18139.107,E2 -18139.107} C_VEL
LIN {X 0,Y 306.892,Z 370.808,A -85,B 0,C 180,E1 -18140.118,E2 -18140.118} C_VEL
LIN {X 0,Y 299.233,Z 384.169,A -85,B 0,C 180,E1 -18142.364,E2 -18142.364} C_VEL
LIN {X 0,Y 292.313,Z 395.736,A -85,B 0,C 180,E1 -18144.759,E2 -18144.759} C_VEL
LIN {X 0,Y 286.147,Z 405.785,A -85,B 0,C 180,E1 -18147.294,E2 -18147.294} C_VEL
LIN {X 0,Y 280.749,Z 414.386,A -85,B 0,C 180,E1 -18149.957,E2 -18149.957} C_VEL
LIN {X 0,Y 276.109,Z 421.66,A -85,B 0,C 180,E1 -18152.731,E2 -18152.731} C_VEL
LIN {X 0,Y 272.126,Z 427.697,A -85,B 0,C 180,E1 -18155.593,E2 -18155.593} C_VEL
LIN {X 0,Y 268.963,Z 432.491,A -85,B 0,C 180,E1 -18158.542,E2 -18158.542} C_VEL
LIN {X 0,Y 265.988,Z 436.593,A -85,B 0,C 180,E1 -18162.028,E2 -18162.028} C_VEL
LIN {X 0,Y 264.383,Z 438.63,A -85,B 0,C 180,E1 -18164.584,E2 -18164.584} C_VEL
LIN {X 0,Y 262.98,Z 439.959,A -85,B 0,C 180,E1 -18167.655,E2 -18167.655} C_VEL
LIN {X 0,Y 262.115,Z 440.124,A -85,B 0,C 180,E1 -18170.743,E2 -18170.743} C_VEL
LIN {X 0,Y 261.641,Z 439.131,A -85,B 0,C 180,E1 -18173.832,E2 -18173.832} C_VEL
LIN {X 0,Y 261.472,Z 436.951,A -85,B 0,C 180,E1 -18176.919,E2 -18176.919} C_VEL
LIN {X 0,Y 261.417,Z 433.548,A -85,B 0,C 180,E1 -18180,E2 -18180} C_VEL
LIN {X 0,Y 261.692,Z 428.823,A -85,B 0,C 180,E1 -18183.079,E2 -18183.079} C_VEL
LIN {X 0,Y 262.415,Z 422.701,A -85,B 0,C 180,E1 -18186.15,E2 -18186.15} C_VEL
LIN {X 0,Y 263.184,Z 415.026,A -85,B 0,C 180,E1 -18189.22,E2 -18189.22} C_VEL
LIN {X 0,Y 264.316,Z 406.849,A -85,B 0,C 180,E1 -18191.892,E2 -18191.892} C_VEL
LIN {X 0,Y 265.879,Z 397.114,A -85,B 0,C 180,E1 -18194.544,E2 -18194.544} C_VEL
LIN {X 0,Y 267.735,Z 385.523,A -85,B 0,C 180,E1 -18197.177,E2 -18197.177} C_VEL
LIN {X 0,Y 269.871,Z 372.724,A -85,B 0,C 180,E1 -18199.591,E2 -18199.591} C_VEL
LIN {X 0,Y 271.884,Z 359.901,A -85,B 0,C 180,E1 -18201.614,E2 -18201.614} C_VEL
LIN {X 0,Y 274.031,Z 346.122,A -85,B 0,C 180,E1 -18203.424,E2 -18203.424} C_VEL
LIN {X 0,Y 275.696,Z 334.112,A -85,B 0,C 180,E1 -18204.739,E2 -18204.739} C_VEL
LIN {X 0,Y 272.558,Z 320.603,A -85,B 0,C 180,E1 -18206.328,E2 -18206.328} C_VEL
LIN {X 0,Y 268.454,Z 305.238,A -85,B 0,C 180,E1 -18207.925,E2 -18207.925} C_VEL
LIN {X 0,Y 264.875,Z 294.003,A -85,B 0,C 180,E1 -18208.998,E2 -18208.998} C_VEL
LIN {X 0,Y 262.609,Z 287.399,A -85,B 0,C 180,E1 -18209.604,E2 -18209.604} C_VEL
LIN {X 0,Y 262.854,Z 287.366,A -85,B 0,C 180,E1 -18212.327,E2 -18212.327} C_VEL
LIN {X 0,Y 263.111,Z 287.335,A -85,B 0,C 180,E1 -18215.991,E2 -18215.991} C_VEL
LIN {X 0,Y 263.108,Z 287.336,A -85,B 0,C 180,E1 -18219.873,E2 -18219.873} C_VEL
LIN {X 0,Y 263.106,Z 287.335,A -85,B 0,C 180,E1 -18223.988,E2 -18223.988} C_VEL
LIN {X 0,Y 263.127,Z 287.332,A -85,B 0,C 180,E1 -18228.407,E2 -18228.407} C_VEL
LIN {X 0,Y 263.184,Z 287.326,A -85,B 0,C 180,E1 -18233.237,E2 -18233.237} C_VEL
LIN {X 0,Y 263.135,Z 287.33,A -85,B 0,C 180,E1 -18237.712,E2 -18237.712} C_VEL
LIN {X 0,Y 263.199,Z 287.323,A -85,B 0,C 180,E1 -18241.785,E2 -18241.785} C_VEL
LIN {X 0,Y 263.228,Z 287.318,A -85,B 0,C 180,E1 -18245.201,E2 -18245.201} C_VEL
LIN {X 0,Y 263.265,Z 287.314,A -85,B 0,C 180,E1 -18249.693,E2 -18249.693} C_VEL
LIN {X 0,Y 263.354,Z 287.304,A -85,B 0,C 180,E1 -18254.522,E2 -18254.522} C_VEL
LIN {X 0,Y 263.358,Z 287.303,A -85,B 0,C 180,E1 -18259.234,E2 -18259.234} C_VEL
LIN {X 0,Y 263.529,Z 287.282,A -85,B 0,C 180,E1 -18262.337,E2 -18262.337} C_VEL
LIN {X 0,Y 263.75,Z 287.255,A -85,B 0,C 180,E1 -18268.473,E2 -18268.473} C_VEL
LIN {X 0,Y 263.751,Z 287.254,A -85,B 0,C 180,E1 -18271.527,E2 -18271.527} C_VEL
LIN {X 0,Y 263.535,Z 287.284,A -85,B 0,C 180,E1 -18277.663,E2 -18277.663} C_VEL
LIN {X 0,Y 263.356,Z 287.302,A -85,B 0,C 180,E1 -18280.766,E2 -18280.766} C_VEL
LIN {X 0,Y 263.354,Z 287.306,A -85,B 0,C 180,E1 -18285.478,E2 -18285.478} C_VEL
LIN {X 0,Y 263.272,Z 287.313,A -85,B 0,C 180,E1 -18290.306,E2 -18290.306} C_VEL
LIN {X 0,Y 263.211,Z 287.324,A -85,B 0,C 180,E1 -18295.291,E2 -18295.291} C_VEL
LIN {X 0,Y 263.169,Z 287.327,A -85,B 0,C 180,E1 -18298.731,E2 -18298.731} C_VEL
LIN {X 0,Y 263.136,Z 287.33,A -85,B 0,C 180,E1 -18302.288,E2 -18302.288} C_VEL
LIN {X 0,Y 263.178,Z 287.326,A -85,B 0,C 180,E1 -18306.761,E2 -18306.761} C_VEL
LIN {X 0,Y 263.094,Z 287.335,A -85,B 0,C 180,E1 -18309.875,E2 -18309.875} C_VEL
LIN {X 0,Y 263.1,Z 287.334,A -85,B 0,C 180,E1 -18313.989,E2 -18313.989} C_VEL
LIN {X 0,Y 263.127,Z 287.332,A -85,B 0,C 180,E1 -18318.406,E2 -18318.406} C_VEL
LIN {X 0,Y 263.185,Z 287.326,A -85,B 0,C 180,E1 -18323.237,E2 -18323.237} C_VEL
LIN {X 0,Y 263.136,Z 287.329,A -85,B 0,C 180,E1 -18327.712,E2 -18327.712} C_VEL
LIN {X 0,Y 263.199,Z 287.322,A -85,B 0,C 180,E1 -18331.785,E2 -18331.785} C_VEL
LIN {X 0,Y 263.229,Z 287.319,A -85,B 0,C 180,E1 -18335.2,E2 -18335.2} C_VEL
LIN {X 0,Y 263.266,Z 287.314,A -85,B 0,C 180,E1 -18339.693,E2 -18339.693} C_VEL
LIN {X 0,Y 263.355,Z 287.304,A -85,B 0,C 180,E1 -18344.522,E2 -18344.522} C_VEL
LIN {X 0,Y 263.356,Z 287.303,A -85,B 0,C 180,E1 -18349.233,E2 -18349.233} C_VEL
LIN {X 0,Y 263.53,Z 287.283,A -85,B 0,C 180,E1 -18352.337,E2 -18352.337} C_VEL
LIN {X 0,Y 263.752,Z 287.255,A -85,B 0,C 180,E1 -18358.473,E2 -18358.473} C_VEL
LIN {X 0,Y 263.752,Z 287.254,A -85,B 0,C 180,E1 -18361.527,E2 -18361.527} C_VEL
LIN {X 0,Y 263.53,Z 287.284,A -85,B 0,C 180,E1 -18367.662,E2 -18367.662} C_VEL
LIN {X 0,Y 263.356,Z 287.301,A -85,B 0,C 180,E1 -18370.766,E2 -18370.766} C_VEL
LIN {X 0,Y 263.354,Z 287.306,A -85,B 0,C 180,E1 -18375.477,E2 -18375.477} C_VEL
LIN {X 0,Y 263.267,Z 287.315,A -85,B 0,C 180,E1 -18380.306,E2 -18380.306} C_VEL
LIN {X 0,Y 263.17,Z 287.331,A -85,B 0,C 180,E1 -18385.295,E2 -18385.295} C_VEL
LIN {X 0,Y 263.213,Z 287.448,A -85,B 0,C 180,E1 -18387.474,E2 -18387.474} C_VEL
LIN {X 0,Y 263.81,Z 291.332,A -85,B 0,C 180,E1 -18391.515,E2 -18391.515} C_VEL
LIN {X 0,Y 264.071,Z 293.274,A -85,B 0,C 180,E1 -18393.439,E2 -18393.439} C_VEL
LIN {X 0,Y 263.644,Z 294.653,A -85,B 0,C 180,E1 -18394.682,E2 -18394.682} C_VEL
LIN {X 0,Y 261.174,Z 297.202,A -85,B 0,C 180,E1 -18396.704,E2 -18396.704} C_VEL
LIN {X 0,Y 259.083,Z 299.292,A -85,B 0,C 180,E1 -18398.345,E2 -18398.345} C_VEL
LIN {X 0,Y 258.328,Z 300.799,A -85,B 0,C 180,E1 -18399.614,E2 -18399.614} C_VEL
LIN {X 0,Y 258.348,Z 301.275,A -85,B 0,C 180,E1 -18400.042,E2 -18400.042} C_VEL
LIN {X 0,Y 259.234,Z 305.412,A -85,B 0,C 180,E1 -18403.761,E2 -18403.761} C_VEL
LIN {X 0,Y 259.629,Z 309.187,A -85,B 0,C 180,E1 -18406.959,E2 -18406.959} C_VEL
LIN {X 0,Y 259.277,Z 312.237,A -85,B 0,C 180,E1 -18409.417,E2 -18409.417} C_VEL
LIN {X 0,Y 258.508,Z 316.089,A -85,B 0,C 180,E1 -18412.436,E2 -18412.436} C_VEL
LIN {X 0,Y 262.254,Z 334.001,A -85,B 0,C 180,E1 -18413.981,E2 -18413.981} C_VEL
LIN {X 0,Y 265.458,Z 350.147,A -85,B 0,C 180,E1 -18415.632,E2 -18415.632} C_VEL
LIN {X 0,Y 268.06,Z 364.885,A -85,B 0,C 180,E1 -18417.367,E2 -18417.367} C_VEL
LIN {X 0,Y 270.282,Z 379.43,A -85,B 0,C 180,E1 -18419.324,E2 -18419.324} C_VEL
LIN {X 0,Y 270.559,Z 383.632,A -85,B 0,C 180,E1 -18419.93,E2 -18419.93} C_VEL
LIN {X 0,Y 267.556,Z 396.743,A -85,B 0,C 180,E1 -18421.783,E2 -18421.783} C_VEL
LIN {X 0,Y 264.653,Z 409.664,A -85,B 0,C 180,E1 -18424.013,E2 -18424.013} C_VEL
LIN {X 0,Y 262.073,Z 420.562,A -85,B 0,C 180,E1 -18426.281,E2 -18426.281} C_VEL
LIN {X 0,Y 259.67,Z 431.364,A -85,B 0,C 180,E1 -18428.985,E2 -18428.985} C_VEL
LIN {X 0,Y 257.71,Z 440.401,A -85,B 0,C 180,E1 -18431.723,E2 -18431.723} C_VEL
LIN {X 0,Y 256.441,Z 446.975,A -85,B 0,C 180,E1 -18434.094,E2 -18434.094} C_VEL
LIN {X 0,Y 255.217,Z 454.226,A -85,B 0,C 180,E1 -18437.273,E2 -18437.273} C_VEL
LIN {X 0,Y 254.599,Z 459.941,A -85,B 0,C 180,E1 -18440.466,E2 -18440.466} C_VEL
LIN {X 0,Y 254.344,Z 464.236,A -85,B 0,C 180,E1 -18443.654,E2 -18443.654} C_VEL
LIN {X 0,Y 254.342,Z 465.887,A -85,B 0,C 180,E1 -18445.245,E2 -18445.245} C_VEL
LIN {X 0,Y 254.214,Z 468.174,A -85,B 0,C 180,E1 -18448.416,E2 -18448.416} C_VEL
LIN {X 0,Y 254.268,Z 468.839,A -85,B 0,C 180,E1 -18450,E2 -18450} C_VEL
LIN {X 0,Y 254.178,Z 469.255,A -85,B 0,C 180,E1 -18453.17,E2 -18453.17} C_VEL
LIN {X 0,Y 254.147,Z 468.52,A -85,B 0,C 180,E1 -18456.351,E2 -18456.351} C_VEL
LIN {X 0,Y 254.381,Z 466.695,A -85,B 0,C 180,E1 -18459.542,E2 -18459.542} C_VEL
LIN {X 0,Y 255.161,Z 463.743,A -85,B 0,C 180,E1 -18462.729,E2 -18462.729} C_VEL
LIN {X 0,Y 256.605,Z 459.77,A -85,B 0,C 180,E1 -18465.896,E2 -18465.896} C_VEL
LIN {X 0,Y 258.76,Z 454.787,A -85,B 0,C 180,E1 -18469.022,E2 -18469.022} C_VEL
LIN {X 0,Y 262.526,Z 447.003,A -85,B 0,C 180,E1 -18472.841,E2 -18472.841} C_VEL
LIN {X 0,Y 266.958,Z 438.59,A -85,B 0,C 180,E1 -18476.166,E2 -18476.166} C_VEL
LIN {X 0,Y 273.273,Z 427.518,A -85,B 0,C 180,E1 -18479.675,E2 -18479.675} C_VEL
LIN {X 0,Y 280.201,Z 415.9,A -85,B 0,C 180,E1 -18482.634,E2 -18482.634} C_VEL
LIN {X 0,Y 287.295,Z 404.118,A -85,B 0,C 180,E1 -18485.091,E2 -18485.091} C_VEL
LIN {X 0,Y 290.65,Z 398.386,A -85,B 0,C 180,E1 -18486.162,E2 -18486.162} C_VEL
LIN {X 0,Y 294.955,Z 389.071,A -85,B 0,C 180,E1 -18488.281,E2 -18488.281} C_VEL
LIN {X 0,Y 297.026,Z 383.841,A -85,B 0,C 180,E1 -18489.707,E2 -18489.707} C_VEL
LIN {X 0,Y 298.648,Z 379.485,A -85,B 0,C 180,E1 -18491.218,E2 -18491.218} C_VEL
LIN {X 0,Y 300.024,Z 375.927,A -85,B 0,C 180,E1 -18492.791,E2 -18492.791} C_VEL
LIN {X 0,Y 300.577,Z 374.668,A -85,B 0,C 180,E1 -18493.545,E2 -18493.545} C_VEL
LIN {X 0,Y 301.12,Z 373.593,A -85,B 0,C 180,E1 -18494.442,E2 -18494.442} C_VEL
LIN {X 0,Y 301.706,Z 372.803,A -85,B 0,C 180,E1 -18495.668,E2 -18495.668} C_VEL
LIN {X 0,Y 302.147,Z 373.329,A -85,B 0,C 180,E1 -18497.582,E2 -18497.582} C_VEL
LIN {X 0,Y 302.268,Z 373.693,A -85,B 0,C 180,E1 -18498.076,E2 -18498.076} C_VEL
LIN {X 0,Y 302.307,Z 375.309,A -85,B 0,C 180,E1 -18499.388,E2 -18499.388} C_VEL
LIN {X 0,Y 294.263,Z 387.9,A -85,B 0,C 180,E1 -18501.613,E2 -18501.613} C_VEL
LIN {X 0,Y 286.299,Z 400.021,A -85,B 0,C 180,E1 -18504.295,E2 -18504.295} C_VEL
LIN {X 0,Y 279.114,Z 410.554,A -85,B 0,C 180,E1 -18507.224,E2 -18507.224} C_VEL
LIN {X 0,Y 273.634,Z 418.405,A -85,B 0,C 180,E1 -18509.945,E2 -18509.945} C_VEL
LIN {X 0,Y 268.302,Z 425.874,A -85,B 0,C 180,E1 -18513.204,E2 -18513.204} C_VEL
LIN {X 0,Y 264.06,Z 431.626,A -85,B 0,C 180,E1 -18516.47,E2 -18516.47} C_VEL
LIN {X 0,Y 260.98,Z 435.597,A -85,B 0,C 180,E1 -18519.508,E2 -18519.508} C_VEL
LIN {X 0,Y 258.565,Z 438.447,A -85,B 0,C 180,E1 -18522.603,E2 -18522.603} C_VEL
LIN {X 0,Y 256.693,Z 440.214,A -85,B 0,C 180,E1 -18525.735,E2 -18525.735} C_VEL
LIN {X 0,Y 255.507,Z 440.832,A -85,B 0,C 180,E1 -18528.899,E2 -18528.899} C_VEL
LIN {X 0,Y 254.781,Z 440.269,A -85,B 0,C 180,E1 -18532.073,E2 -18532.073} C_VEL
LIN {X 0,Y 254.463,Z 438.538,A -85,B 0,C 180,E1 -18535.248,E2 -18535.248} C_VEL
LIN {X 0,Y 254.344,Z 435.616,A -85,B 0,C 180,E1 -18538.417,E2 -18538.417} C_VEL
LIN {X 0,Y 254.409,Z 431.435,A -85,B 0,C 180,E1 -18541.583,E2 -18541.583} C_VEL
LIN {X 0,Y 254.971,Z 425.89,A -85,B 0,C 180,E1 -18544.744,E2 -18544.744} C_VEL
LIN {X 0,Y 255.515,Z 420.796,A -85,B 0,C 180,E1 -18547.11,E2 -18547.11} C_VEL
LIN {X 0,Y 256.424,Z 412.534,A -85,B 0,C 180,E1 -18550.262,E2 -18550.262} C_VEL
LIN {X 0,Y 258.026,Z 402.421,A -85,B 0,C 180,E1 -18553.387,E2 -18553.387} C_VEL
LIN {X 0,Y 259.756,Z 391.772,A -85,B 0,C 180,E1 -18556.101,E2 -18556.101} C_VEL
LIN {X 0,Y 261.944,Z 379.052,A -85,B 0,C 180,E1 -18558.782,E2 -18558.782} C_VEL
LIN {X 0,Y 264.248,Z 365.234,A -85,B 0,C 180,E1 -18561.192,E2 -18561.192} C_VEL
LIN {X 0,Y 266.286,Z 351.956,A -85,B 0,C 180,E1 -18563.116,E2 -18563.116} C_VEL
LIN {X 0,Y 268.642,Z 337.063,A -85,B 0,C 180,E1 -18564.881,E2 -18564.881} C_VEL
LIN {X 0,Y 268.73,Z 334.686,A -85,B 0,C 180,E1 -18565.143,E2 -18565.143} C_VEL
LIN {X 0,Y 265.066,Z 319.223,A -85,B 0,C 180,E1 -18567.007,E2 -18567.007} C_VEL
LIN {X 0,Y 260.571,Z 302.622,A -85,B 0,C 180,E1 -18568.769,E2 -18568.769} C_VEL
LIN {X 0,Y 255.613,Z 288.268,A -85,B 0,C 180,E1 -18570.169,E2 -18570.169} C_VEL
LIN {X 0,Y 255.952,Z 288.226,A -85,B 0,C 180,E1 -18574.538,E2 -18574.538} C_VEL
LIN {X 0,Y 256.089,Z 288.214,A -85,B 0,C 180,E1 -18577.262,E2 -18577.262} C_VEL
LIN {X 0,Y 256.057,Z 288.217,A -85,B 0,C 180,E1 -18581.203,E2 -18581.203} C_VEL
LIN {X 0,Y 256.044,Z 288.216,A -85,B 0,C 180,E1 -18585.534,E2 -18585.534} C_VEL
LIN {X 0,Y 256.057,Z 288.216,A -85,B 0,C 180,E1 -18588.797,E2 -18588.797} C_VEL
LIN {X 0,Y 256.133,Z 288.207,A -85,B 0,C 180,E1 -18592.868,E2 -18592.868} C_VEL
LIN {X 0,Y 256.07,Z 288.215,A -85,B 0,C 180,E1 -18596.707,E2 -18596.707} C_VEL
LIN {X 0,Y 256.106,Z 288.209,A -85,B 0,C 180,E1 -18600.399,E2 -18600.399} C_VEL
LIN {X 0,Y 256.191,Z 288.196,A -85,B 0,C 180,E1 -18604.862,E2 -18604.862} C_VEL
LIN {X 0,Y 256.167,Z 288.199,A -85,B 0,C 180,E1 -18609.105,E2 -18609.105} C_VEL
LIN {X 0,Y 256.303,Z 288.183,A -85,B 0,C 180,E1 -18614.085,E2 -18614.085} C_VEL
LIN {X 0,Y 256.298,Z 288.182,A -85,B 0,C 180,E1 -18617.328,E2 -18617.328} C_VEL
LIN {X 0,Y 256.437,Z 288.166,A -85,B 0,C 180,E1 -18620.623,E2 -18620.623} C_VEL
LIN {X 0,Y 256.46,Z 288.161,A -85,B 0,C 180,E1 -18623.707,E2 -18623.707} C_VEL
LIN {X 0,Y 256.713,Z 288.131,A -85,B 0,C 180,E1 -18628.431,E2 -18628.431} C_VEL
LIN {X 0,Y 256.714,Z 288.13,A -85,B 0,C 180,E1 -18631.569,E2 -18631.569} C_VEL
LIN {X 0,Y 256.465,Z 288.162,A -85,B 0,C 180,E1 -18636.293,E2 -18636.293} C_VEL
LIN {X 0,Y 256.43,Z 288.166,A -85,B 0,C 180,E1 -18639.465,E2 -18639.465} C_VEL
LIN {X 0,Y 256.258,Z 288.188,A -85,B 0,C 180,E1 -18644.29,E2 -18644.29} C_VEL
LIN {X 0,Y 256.214,Z 288.195,A -85,B 0,C 180,E1 -18647.562,E2 -18647.562} C_VEL
LIN {X 0,Y 256.189,Z 288.197,A -85,B 0,C 180,E1 -18651.136,E2 -18651.136} C_VEL
LIN {X 0,Y 256.191,Z 288.197,A -85,B 0,C 180,E1 -18655.138,E2 -18655.138} C_VEL
LIN {X 0,Y 256.107,Z 288.208,A -85,B 0,C 180,E1 -18659.601,E2 -18659.601} C_VEL
LIN {X 0,Y 256.071,Z 288.212,A -85,B 0,C 180,E1 -18663.293,E2 -18663.293} C_VEL
LIN {X 0,Y 256.113,Z 288.209,A -85,B 0,C 180,E1 -18667.269,E2 -18667.269} C_VEL
LIN {X 0,Y 256.021,Z 288.218,A -85,B 0,C 180,E1 -18671.21,E2 -18671.21} C_VEL
LIN {X 0,Y 256.042,Z 288.215,A -85,B 0,C 180,E1 -18675.534,E2 -18675.534} C_VEL
LIN {X 0,Y 256.058,Z 288.216,A -85,B 0,C 180,E1 -18678.797,E2 -18678.797} C_VEL
LIN {X 0,Y 256.133,Z 288.207,A -85,B 0,C 180,E1 -18682.867,E2 -18682.867} C_VEL
LIN {X 0,Y 256.071,Z 288.214,A -85,B 0,C 180,E1 -18686.707,E2 -18686.707} C_VEL
LIN {X 0,Y 256.107,Z 288.207,A -85,B 0,C 180,E1 -18690.399,E2 -18690.399} C_VEL
LIN {X 0,Y 256.191,Z 288.197,A -85,B 0,C 180,E1 -18694.862,E2 -18694.862} C_VEL
LIN {X 0,Y 256.168,Z 288.198,A -85,B 0,C 180,E1 -18699.105,E2 -18699.105} C_VEL
LIN {X 0,Y 256.304,Z 288.183,A -85,B 0,C 180,E1 -18704.085,E2 -18704.085} C_VEL
LIN {X 0,Y 256.299,Z 288.182,A -85,B 0,C 180,E1 -18708.933,E2 -18708.933} C_VEL
LIN {X 0,Y 256.493,Z 288.161,A -85,B 0,C 180,E1 -18712.125,E2 -18712.125} C_VEL
LIN {X 0,Y 256.493,Z 288.158,A -85,B 0,C 180,E1 -18716.858,E2 -18716.858} C_VEL
LIN {X 0,Y 256.747,Z 288.13,A -85,B 0,C 180,E1 -18720,E2 -18720} C_VEL
LIN {X 0,Y 256.498,Z 288.156,A -85,B 0,C 180,E1 -18723.141,E2 -18723.141} C_VEL
LIN {X 0,Y 256.494,Z 288.161,A -85,B 0,C 180,E1 -18727.874,E2 -18727.874} C_VEL
LIN {X 0,Y 256.299,Z 288.181,A -85,B 0,C 180,E1 -18731.066,E2 -18731.066} C_VEL
LIN {X 0,Y 256.303,Z 288.183,A -85,B 0,C 180,E1 -18735.914,E2 -18735.914} C_VEL
LIN {X 0,Y 256.169,Z 288.199,A -85,B 0,C 180,E1 -18740.895,E2 -18740.895} C_VEL
LIN {X 0,Y 256.135,Z 288.206,A -85,B 0,C 180,E1 -18745.112,E2 -18745.112} C_VEL
LIN {X 0,Y 256.186,Z 288.361,A -85,B 0,C 180,E1 -18747.134,E2 -18747.134} C_VEL
LIN {X 0,Y 256.772,Z 292.317,A -85,B 0,C 180,E1 -18751.335,E2 -18751.335} C_VEL
LIN {X 0,Y 257.345,Z 295.955,A -85,B 0,C 180,E1 -18754.994,E2 -18754.994} C_VEL
LIN {X 0,Y 258.105,Z 299.895,A -85,B 0,C 180,E1 -18758.775,E2 -18758.775} C_VEL
LIN {X 0,Y 258.348,Z 301.275,A -85,B 0,C 180,E1 -18760.042,E2 -18760.042} C_VEL
LIN {X 0,Y 257.999,Z 302.751,A -85,B 0,C 180,E1 -18761.308,E2 -18761.308} C_VEL
LIN {X 0,Y 255.635,Z 305.408,A -85,B 0,C 180,E1 -18763.373,E2 -18763.373} C_VEL
LIN {X 0,Y 252.796,Z 308.671,A -85,B 0,C 180,E1 -18765.905,E2 -18765.905} C_VEL
LIN {X 0,Y 252.537,Z 309.721,A -85,B 0,C 180,E1 -18766.778,E2 -18766.778} C_VEL
LIN {X 0,Y 252.368,Z 312.1,A -85,B 0,C 180,E1 -18768.755,E2 -18768.755} C_VEL
LIN {X 0,Y 251.591,Z 315.845,A -85,B 0,C 180,E1 -18771.727,E2 -18771.727} C_VEL
LIN {X 0,Y 255.297,Z 333.918,A -85,B 0,C 180,E1 -18773.335,E2 -18773.335} C_VEL
LIN {X 0,Y 258.448,Z 350.035,A -85,B 0,C 180,E1 -18775.037,E2 -18775.037} C_VEL
LIN {X 0,Y 261.235,Z 366.06,A -85,B 0,C 180,E1 -18777.002,E2 -18777.002} C_VEL
LIN {X 0,Y 263.429,Z 380.981,A -85,B 0,C 180,E1 -18779.108,E2 -18779.108} C_VEL
LIN {X 0,Y 263.645,Z 384.083,A -85,B 0,C 180,E1 -18779.57,E2 -18779.57} C_VEL
LIN {X 0,Y 260.448,Z 397.82,A -85,B 0,C 180,E1 -18781.601,E2 -18781.601} C_VEL
LIN {X 0,Y 257.708,Z 409.459,A -85,B 0,C 180,E1 -18783.694,E2 -18783.694} C_VEL
LIN {X 0,Y 255.079,Z 420.312,A -85,B 0,C 180,E1 -18786.021,E2 -18786.021} C_VEL
LIN {X 0,Y 252.642,Z 431.066,A -85,B 0,C 180,E1 -18788.799,E2 -18788.799} C_VEL
LIN {X 0,Y 250.637,Z 440.05,A -85,B 0,C 180,E1 -18791.611,E2 -18791.611} C_VEL
LIN {X 0,Y 249.143,Z 447.571,A -85,B 0,C 180,E1 -18794.456,E2 -18794.456} C_VEL
LIN {X 0,Y 248.014,Z 454.594,A -85,B 0,C 180,E1 -18797.729,E2 -18797.729} C_VEL
LIN {X 0,Y 247.473,Z 460.1,A -85,B 0,C 180,E1 -18801.014,E2 -18801.014} C_VEL
LIN {X 0,Y 247.309,Z 463.947,A -85,B 0,C 180,E1 -18804.055,E2 -18804.055} C_VEL
LIN {X 0,Y 247.158,Z 466.376,A -85,B 0,C 180,E1 -18806.74,E2 -18806.74} C_VEL
LIN {X 0,Y 247.198,Z 468.161,A -85,B 0,C 180,E1 -18810,E2 -18810} C_VEL
LIN {X 0,Y 247.107,Z 468.73,A -85,B 0,C 180,E1 -18813.261,E2 -18813.261} C_VEL
LIN {X 0,Y 247.054,Z 468.159,A -85,B 0,C 180,E1 -18816.534,E2 -18816.534} C_VEL
LIN {X 0,Y 247.33,Z 466.429,A -85,B 0,C 180,E1 -18819.817,E2 -18819.817} C_VEL
LIN {X 0,Y 248.195,Z 463.677,A -85,B 0,C 180,E1 -18823.093,E2 -18823.093} C_VEL
LIN {X 0,Y 249.732,Z 459.941,A -85,B 0,C 180,E1 -18826.345,E2 -18826.345} C_VEL
LIN {X 0,Y 252.716,Z 453.8,A -85,B 0,C 180,E1 -18830.342,E2 -18830.342} C_VEL
LIN {X 0,Y 256.934,Z 446.067,A -85,B 0,C 180,E1 -18834.224,E2 -18834.224} C_VEL
LIN {X 0,Y 261.982,Z 437.622,A -85,B 0,C 180,E1 -18837.613,E2 -18837.613} C_VEL
LIN {X 0,Y 268.069,Z 428.025,A -85,B 0,C 180,E1 -18840.746,E2 -18840.746} C_VEL
LIN {X 0,Y 274.501,Z 418.198,A -85,B 0,C 180,E1 -18843.399,E2 -18843.399} C_VEL
LIN {X 0,Y 282.846,Z 405.551,A -85,B 0,C 180,E1 -18846.166,E2 -18846.166} C_VEL
LIN {X 0,Y 285.788,Z 401.028,A -85,B 0,C 180,E1 -18847.049,E2 -18847.049} C_VEL
LIN {X 0,Y 290.199,Z 392.745,A -85,B 0,C 180,E1 -18849.026,E2 -18849.026} C_VEL
LIN {X 0,Y 292.543,Z 387.833,A -85,B 0,C 180,E1 -18850.44,E2 -18850.44} C_VEL
LIN {X 0,Y 294.784,Z 382.863,A -85,B 0,C 180,E1 -18852.348,E2 -18852.348} C_VEL
LIN {X 0,Y 295.926,Z 380.585,A -85,B 0,C 180,E1 -18853.53,E2 -18853.53} C_VEL
LIN {X 0,Y 296.826,Z 379.032,A -85,B 0,C 180,E1 -18854.74,E2 -18854.74} C_VEL
LIN {X 0,Y 297.055,Z 378.725,A -85,B 0,C 180,E1 -18855.216,E2 -18855.216} C_VEL
LIN {X 0,Y 297.579,Z 378.654,A -85,B 0,C 180,E1 -18857.066,E2 -18857.066} C_VEL
LIN {X 0,Y 297.674,Z 379.924,A -85,B 0,C 180,E1 -18858.619,E2 -18858.619} C_VEL
LIN {X 0,Y 289.355,Z 391.726,A -85,B 0,C 180,E1 -18860.839,E2 -18860.839} C_VEL
LIN {X 0,Y 281.05,Z 403.076,A -85,B 0,C 180,E1 -18863.522,E2 -18863.522} C_VEL
LIN {X 0,Y 273.555,Z 413.043,A -85,B 0,C 180,E1 -18866.471,E2 -18866.471} C_VEL
LIN {X 0,Y 267.791,Z 420.494,A -85,B 0,C 180,E1 -18869.219,E2 -18869.219} C_VEL
LIN {X 0,Y 262.465,Z 427.224,A -85,B 0,C 180,E1 -18872.336,E2 -18872.336} C_VEL
LIN {X 0,Y 258.547,Z 431.93,A -85,B 0,C 180,E1 -18875.082,E2 -18875.082} C_VEL
LIN {X 0,Y 255.956,Z 435.057,A -85,B 0,C 180,E1 -18877.393,E2 -18877.393} C_VEL
LIN {X 0,Y 252.514,Z 438.753,A -85,B 0,C 180,E1 -18881.138,E2 -18881.138} C_VEL
LIN {X 0,Y 250.739,Z 440.329,A -85,B 0,C 180,E1 -18883.723,E2 -18883.723} C_VEL
LIN {X 0,Y 249.105,Z 441.34,A -85,B 0,C 180,E1 -18886.956,E2 -18886.956} C_VEL
LIN {X 0,Y 248.082,Z 441.234,A -85,B 0,C 180,E1 -18890.214,E2 -18890.214} C_VEL
LIN {X 0,Y 247.53,Z 439.9,A -85,B 0,C 180,E1 -18893.588,E2 -18893.588} C_VEL
LIN {X 0,Y 247.309,Z 437.494,A -85,B 0,C 180,E1 -18896.742,E2 -18896.742} C_VEL
LIN {X 0,Y 247.252,Z 433.802,A -85,B 0,C 180,E1 -18900,E2 -18900} C_VEL
LIN {X 0,Y 247.558,Z 428.811,A -85,B 0,C 180,E1 -18903.255,E2 -18903.255} C_VEL
LIN {X 0,Y 248.301,Z 422.42,A -85,B 0,C 180,E1 -18906.501,E2 -18906.501} C_VEL
LIN {X 0,Y 249.159,Z 414.419,A -85,B 0,C 180,E1 -18909.744,E2 -18909.744} C_VEL
LIN {X 0,Y 250.627,Z 404.639,A -85,B 0,C 180,E1 -18912.964,E2 -18912.964} C_VEL
LIN {X 0,Y 252.369,Z 394.351,A -85,B 0,C 180,E1 -18915.755,E2 -18915.755} C_VEL
LIN {X 0,Y 254.458,Z 382.07,A -85,B 0,C 180,E1 -18918.52,E2 -18918.52} C_VEL
LIN {X 0,Y 256.692,Z 369.618,A -85,B 0,C 180,E1 -18920.851,E2 -18920.851} C_VEL
LIN {X 0,Y 258.842,Z 356.035,A -85,B 0,C 180,E1 -18922.974,E2 -18922.974} C_VEL
LIN {X 0,Y 261.199,Z 341.342,A -85,B 0,C 180,E1 -18924.861,E2 -18924.861} C_VEL
LIN {X 0,Y 261.94,Z 336.346,A -85,B 0,C 180,E1 -18925.423,E2 -18925.423} C_VEL
LIN {X 0,Y 258.48,Z 321.447,A -85,B 0,C 180,E1 -18927.302,E2 -18927.302} C_VEL
LIN {X 0,Y 254.097,Z 305.018,A -85,B 0,C 180,E1 -18929.131,E2 -18929.131} C_VEL
LIN {X 0,Y 248.631,Z 289.139,A -85,B 0,C 180,E1 -18930.756,E2 -18930.756} C_VEL
LIN {X 0,Y 248.948,Z 289.102,A -85,B 0,C 180,E1 -18935.045,E2 -18935.045} C_VEL
LIN {X 0,Y 249.018,Z 289.092,A -85,B 0,C 180,E1 -18938.383,E2 -18938.383} C_VEL
LIN {X 0,Y 249.004,Z 289.096,A -85,B 0,C 180,E1 -18942.791,E2 -18942.791} C_VEL
LIN {X 0,Y 249.012,Z 289.091,A -85,B 0,C 180,E1 -18947.362,E2 -18947.362} C_VEL
LIN {X 0,Y 249.028,Z 289.088,A -85,B 0,C 180,E1 -18951.62,E2 -18951.62} C_VEL
LIN {X 0,Y 249.046,Z 289.086,A -85,B 0,C 180,E1 -18955.64,E2 -18955.64} C_VEL
LIN {X 0,Y 249.05,Z 289.085,A -85,B 0,C 180,E1 -18959.473,E2 -18959.473} C_VEL
LIN {X 0,Y 249.074,Z 289.082,A -85,B 0,C 180,E1 -18963.162,E2 -18963.162} C_VEL
LIN {X 0,Y 249.08,Z 289.082,A -85,B 0,C 180,E1 -18966.733,E2 -18966.733} C_VEL
LIN {X 0,Y 249.112,Z 289.08,A -85,B 0,C 180,E1 -18970.212,E2 -18970.212} C_VEL
LIN {X 0,Y 249.245,Z 289.06,A -85,B 0,C 180,E1 -18973.622,E2 -18973.622} C_VEL
LIN {X 0,Y 249.248,Z 289.062,A -85,B 0,C 180,E1 -18978.616,E2 -18978.616} C_VEL
LIN {X 0,Y 249.438,Z 289.039,A -85,B 0,C 180,E1 -18981.901,E2 -18981.901} C_VEL
LIN {X 0,Y 249.276,Z 289.056,A -85,B 0,C 180,E1 -18985.148,E2 -18985.148} C_VEL
LIN {X 0,Y 249.674,Z 289.008,A -85,B 0,C 180,E1 -18988.387,E2 -18988.387} C_VEL
LIN {X 0,Y 249.676,Z 289.007,A -85,B 0,C 180,E1 -18991.613,E2 -18991.613} C_VEL
LIN {X 0,Y 249.438,Z 289.037,A -85,B 0,C 180,E1 -18996.471,E2 -18996.471} C_VEL
LIN {X 0,Y 249.346,Z 289.05,A -85,B 0,C 180,E1 -18999.736,E2 -18999.736} C_VEL
LIN {X 0,Y 249.209,Z 289.065,A -85,B 0,C 180,E1 -19004.703,E2 -19004.703} C_VEL
LIN {X 0,Y 249.143,Z 289.073,A -85,B 0,C 180,E1 -19008.077,E2 -19008.077} C_VEL
LIN {X 0,Y 249.108,Z 289.082,A -85,B 0,C 180,E1 -19011.516,E2 -19011.516} C_VEL
LIN {X 0,Y 249.134,Z 289.076,A -85,B 0,C 180,E1 -19015.482,E2 -19015.482} C_VEL
LIN {X 0,Y 249.076,Z 289.083,A -85,B 0,C 180,E1 -19018.989,E2 -19018.989} C_VEL
LIN {X 0,Y 249.034,Z 289.087,A -85,B 0,C 180,E1 -19022.426,E2 -19022.426} C_VEL
LIN {X 0,Y 249.029,Z 289.087,A -85,B 0,C 180,E1 -19026.346,E2 -19026.346} C_VEL
LIN {X 0,Y 248.981,Z 289.094,A -85,B 0,C 180,E1 -19030.483,E2 -19030.483} C_VEL
LIN {X 0,Y 248.986,Z 289.096,A -85,B 0,C 180,E1 -19034.884,E2 -19034.884} C_VEL
LIN {X 0,Y 249.012,Z 289.091,A -85,B 0,C 180,E1 -19037.361,E2 -19037.361} C_VEL
LIN {X 0,Y 249.029,Z 289.087,A -85,B 0,C 180,E1 -19041.619,E2 -19041.619} C_VEL
LIN {X 0,Y 249.047,Z 289.085,A -85,B 0,C 180,E1 -19045.639,E2 -19045.639} C_VEL
LIN {X 0,Y 249.051,Z 289.083,A -85,B 0,C 180,E1 -19049.472,E2 -19049.472} C_VEL
LIN {X 0,Y 249.075,Z 289.083,A -85,B 0,C 180,E1 -19053.162,E2 -19053.162} C_VEL
LIN {X 0,Y 249.081,Z 289.082,A -85,B 0,C 180,E1 -19056.732,E2 -19056.732} C_VEL
LIN {X 0,Y 249.114,Z 289.079,A -85,B 0,C 180,E1 -19060.211,E2 -19060.211} C_VEL
LIN {X 0,Y 249.246,Z 289.06,A -85,B 0,C 180,E1 -19063.622,E2 -19063.622} C_VEL
LIN {X 0,Y 249.247,Z 289.062,A -85,B 0,C 180,E1 -19068.616,E2 -19068.616} C_VEL
LIN {X 0,Y 249.438,Z 289.039,A -85,B 0,C 180,E1 -19071.901,E2 -19071.901} C_VEL
LIN {X 0,Y 249.429,Z 289.038,A -85,B 0,C 180,E1 -19076.769,E2 -19076.769} C_VEL
LIN {X 0,Y 249.676,Z 289.009,A -85,B 0,C 180,E1 -19078.387,E2 -19078.387} C_VEL
LIN {X 0,Y 249.677,Z 289.007,A -85,B 0,C 180,E1 -19081.613,E2 -19081.613} C_VEL
LIN {X 0,Y 249.436,Z 289.038,A -85,B 0,C 180,E1 -19086.471,E2 -19086.471} C_VEL
LIN {X 0,Y 249.346,Z 289.05,A -85,B 0,C 180,E1 -19089.736,E2 -19089.736} C_VEL
LIN {X 0,Y 249.208,Z 289.065,A -85,B 0,C 180,E1 -19094.703,E2 -19094.703} C_VEL
LIN {X 0,Y 249.142,Z 289.073,A -85,B 0,C 180,E1 -19098.077,E2 -19098.077} C_VEL
LIN {X 0,Y 249.088,Z 289.085,A -85,B 0,C 180,E1 -19101.518,E2 -19101.518} C_VEL
LIN {X 0,Y 249.1,Z 289.083,A -85,B 0,C 180,E1 -19106.445,E2 -19106.445} C_VEL
LIN {X 0,Y 249.611,Z 292.617,A -85,B 0,C 180,E1 -19110.451,E2 -19110.451} C_VEL
LIN {X 0,Y 250.166,Z 296.216,A -85,B 0,C 180,E1 -19114.185,E2 -19114.185} C_VEL
LIN {X 0,Y 250.964,Z 300.444,A -85,B 0,C 180,E1 -19118.361,E2 -19118.361} C_VEL
LIN {X 0,Y 251.807,Z 304.373,A -85,B 0,C 180,E1 -19122.055,E2 -19122.055} C_VEL
LIN {X 0,Y 252.404,Z 307.681,A -85,B 0,C 180,E1 -19125.013,E2 -19125.013} C_VEL
LIN {X 0,Y 252.537,Z 309.721,A -85,B 0,C 180,E1 -19126.778,E2 -19126.778} C_VEL
LIN {X 0,Y 251.819,Z 310.329,A -85,B 0,C 180,E1 -19127.228,E2 -19127.228} C_VEL
LIN {X 0,Y 249.012,Z 311.295,A -85,B 0,C 180,E1 -19127.805,E2 -19127.805} C_VEL
LIN {X 0,Y 245.873,Z 312.363,A -85,B 0,C 180,E1 -19128.462,E2 -19128.462} C_VEL
LIN {X 0,Y 245.242,Z 312.885,A -85,B 0,C 180,E1 -19128.859,E2 -19128.859} C_VEL
LIN {X 0,Y 244.661,Z 315.452,A -85,B 0,C 180,E1 -19130.98,E2 -19130.98} C_VEL
LIN {X 0,Y 248.334,Z 333.666,A -85,B 0,C 180,E1 -19132.658,E2 -19132.658} C_VEL
LIN {X 0,Y 251.525,Z 350.254,A -85,B 0,C 180,E1 -19134.468,E2 -19134.468} C_VEL
LIN {X 0,Y 254.102,Z 365.586,A -85,B 0,C 180,E1 -19136.415,E2 -19136.415} C_VEL
LIN {X 0,Y 256.32,Z 380.647,A -85,B 0,C 180,E1 -19138.603,E2 -19138.603} C_VEL
LIN {X 0,Y 256.748,Z 383.935,A -85,B 0,C 180,E1 -19139.119,E2 -19139.119} C_VEL
LIN {X 0,Y 253.592,Z 397.604,A -85,B 0,C 180,E1 -19141.215,E2 -19141.215} C_VEL
LIN {X 0,Y 250.453,Z 410.527,A -85,B 0,C 180,E1 -19143.632,E2 -19143.632} C_VEL
LIN {X 0,Y 247.721,Z 421.645,A -85,B 0,C 180,E1 -19146.154,E2 -19146.154} C_VEL
LIN {X 0,Y 245.263,Z 432.074,A -85,B 0,C 180,E1 -19149.011,E2 -19149.011} C_VEL
LIN {X 0,Y 243.161,Z 441.817,A -85,B 0,C 180,E1 -19152.286,E2 -19152.286} C_VEL
LIN {X 0,Y 241.916,Z 448.114,A -85,B 0,C 180,E1 -19154.843,E2 -19154.843} C_VEL
LIN {X 0,Y 240.84,Z 454.907,A -85,B 0,C 180,E1 -19158.213,E2 -19158.213} C_VEL
LIN {X 0,Y 240.346,Z 460.204,A -85,B 0,C 180,E1 -19161.593,E2 -19161.593} C_VEL
LIN {X 0,Y 240.245,Z 464.096,A -85,B 0,C 180,E1 -19164.965,E2 -19164.965} C_VEL
LIN {X 0,Y 240.081,Z 466.649,A -85,B 0,C 180,E1 -19168.322,E2 -19168.322} C_VEL
LIN {X 0,Y 240.13,Z 467.468,A -85,B 0,C 180,E1 -19170,E2 -19170} C_VEL
LIN {X 0,Y 240.037,Z 468.2,A -85,B 0,C 180,E1 -19173.357,E2 -19173.357} C_VEL
LIN {X 0,Y 239.971,Z 467.723,A -85,B 0,C 180,E1 -19176.727,E2 -19176.727} C_VEL
LIN {X 0,Y 240.295,Z 466.175,A -85,B 0,C 180,E1 -19180.107,E2 -19180.107} C_VEL
LIN {X 0,Y 241.24,Z 463.64,A -85,B 0,C 180,E1 -19183.477,E2 -19183.477} C_VEL
LIN {X 0,Y 243.387,Z 459.029,A -85,B 0,C 180,E1 -19187.656,E2 -19187.656} C_VEL
LIN {X 0,Y 246.839,Z 452.899,A -85,B 0,C 180,E1 -19191.724,E2 -19191.724} C_VEL
LIN {X 0,Y 251.602,Z 445.239,A -85,B 0,C 180,E1 -19195.656,E2 -19195.656} C_VEL
LIN {X 0,Y 255.953,Z 438.682,A -85,B 0,C 180,E1 -19198.416,E2 -19198.416} C_VEL
LIN {X 0,Y 262.975,Z 428.682,A -85,B 0,C 180,E1 -19201.858,E2 -19201.858} C_VEL
LIN {X 0,Y 270.706,Z 417.948,A -85,B 0,C 180,E1 -19204.831,E2 -19204.831} C_VEL
LIN {X 0,Y 278.523,Z 407.137,A -85,B 0,C 180,E1 -19207.272,E2 -19207.272} C_VEL
LIN {X 0,Y 281.517,Z 402.853,A -85,B 0,C 180,E1 -19208.162,E2 -19208.162} C_VEL
LIN {X 0,Y 286.07,Z 395.3,A -85,B 0,C 180,E1 -19210.1,E2 -19210.1} C_VEL
LIN {X 0,Y 288.666,Z 390.618,A -85,B 0,C 180,E1 -19211.636,E2 -19211.636} C_VEL
LIN {X 0,Y 290.098,Z 388.005,A -85,B 0,C 180,E1 -19212.714,E2 -19212.714} C_VEL
LIN {X 0,Y 291.12,Z 386.266,A -85,B 0,C 180,E1 -19213.595,E2 -19213.595} C_VEL
LIN {X 0,Y 291.755,Z 385.24,A -85,B 0,C 180,E1 -19214.313,E2 -19214.313} C_VEL
LIN {X 0,Y 292.719,Z 384.047,A -85,B 0,C 180,E1 -19216.078,E2 -19216.078} C_VEL
LIN {X 0,Y 292.915,Z 384.638,A -85,B 0,C 180,E1 -19217.793,E2 -19217.793} C_VEL
LIN {X 0,Y 290.895,Z 387.382,A -85,B 0,C 180,E1 -19218.364,E2 -19218.364} C_VEL
LIN {X 0,Y 281.404,Z 399.397,A -85,B 0,C 180,E1 -19220.952,E2 -19220.952} C_VEL
LIN {X 0,Y 272.236,Z 410.649,A -85,B 0,C 180,E1 -19224.034,E2 -19224.034} C_VEL
LIN {X 0,Y 264.945,Z 419.265,A -85,B 0,C 180,E1 -19227.059,E2 -19227.059} C_VEL
LIN {X 0,Y 259.31,Z 425.766,A -85,B 0,C 180,E1 -19229.908,E2 -19229.908} C_VEL
LIN {X 0,Y 254.436,Z 431.149,A -85,B 0,C 180,E1 -19232.886,E2 -19232.886} C_VEL
LIN {X 0,Y 251.319,Z 434.469,A -85,B 0,C 180,E1 -19235.199,E2 -19235.199} C_VEL
LIN {X 0,Y 247.86,Z 437.977,A -85,B 0,C 180,E1 -19238.37,E2 -19238.37} C_VEL
LIN {X 0,Y 245.072,Z 440.392,A -85,B 0,C 180,E1 -19241.612,E2 -19241.612} C_VEL
LIN {X 0,Y 242.926,Z 441.753,A -85,B 0,C 180,E1 -19244.908,E2 -19244.908} C_VEL
LIN {X 0,Y 241.533,Z 442.013,A -85,B 0,C 180,E1 -19248.248,E2 -19248.248} C_VEL
LIN {X 0,Y 240.681,Z 441.165,A -85,B 0,C 180,E1 -19251.605,E2 -19251.605} C_VEL
LIN {X 0,Y 240.29,Z 439.175,A -85,B 0,C 180,E1 -19254.967,E2 -19254.967} C_VEL
LIN {X 0,Y 240.188,Z 435.969,A -85,B 0,C 180,E1 -19258.324,E2 -19258.324} C_VEL
LIN {X 0,Y 240.257,Z 431.501,A -85,B 0,C 180,E1 -19261.677,E2 -19261.677} C_VEL
LIN {X 0,Y 240.854,Z 425.658,A -85,B 0,C 180,E1 -19265.022,E2 -19265.022} C_VEL
LIN {X 0,Y 241.435,Z 419.578,A -85,B 0,C 180,E1 -19267.836,E2 -19267.836} C_VEL
LIN {X 0,Y 242.442,Z 411.719,A -85,B 0,C 180,E1 -19270.861,E2 -19270.861} C_VEL
LIN {X 0,Y 243.936,Z 402.666,A -85,B 0,C 180,E1 -19273.751,E2 -19273.751} C_VEL
LIN {X 0,Y 245.741,Z 391.894,A -85,B 0,C 180,E1 -19276.619,E2 -19276.619} C_VEL
LIN {X 0,Y 247.708,Z 381.05,A -85,B 0,C 180,E1 -19279.044,E2 -19279.044} C_VEL
LIN {X 0,Y 250,Z 368.349,A -85,B 0,C 180,E1 -19281.436,E2 -19281.436} C_VEL
LIN {X 0,Y 252.271,Z 354.573,A -85,B 0,C 180,E1 -19283.608,E2 -19283.608} C_VEL
LIN {X 0,Y 254.766,Z 339.679,A -85,B 0,C 180,E1 -19285.534,E2 -19285.534} C_VEL
LIN {X 0,Y 255.038,Z 338.019,A -85,B 0,C 180,E1 -19285.723,E2 -19285.723} C_VEL
LIN {X 0,Y 252.277,Z 325.427,A -85,B 0,C 180,E1 -19287.379,E2 -19287.379} C_VEL
LIN {X 0,Y 248.47,Z 310.626,A -85,B 0,C 180,E1 -19289.132,E2 -19289.132} C_VEL
LIN {X 0,Y 243.57,Z 296.024,A -85,B 0,C 180,E1 -19290.736,E2 -19290.736} C_VEL
LIN {X 0,Y 241.653,Z 290.01,A -85,B 0,C 180,E1 -19291.334,E2 -19291.334} C_VEL
LIN {X 0,Y 241.905,Z 289.979,A -85,B 0,C 180,E1 -19295.563,E2 -19295.563} C_VEL
LIN {X 0,Y 241.956,Z 289.973,A -85,B 0,C 180,E1 -19299.72,E2 -19299.72} C_VEL
LIN {X 0,Y 241.921,Z 289.975,A -85,B 0,C 180,E1 -19304.205,E2 -19304.205} C_VEL
LIN {X 0,Y 241.936,Z 289.971,A -85,B 0,C 180,E1 -19308.077,E2 -19308.077} C_VEL
LIN {X 0,Y 241.989,Z 289.967,A -85,B 0,C 180,E1 -19312.418,E2 -19312.418} C_VEL
LIN {X 0,Y 241.983,Z 289.968,A -85,B 0,C 180,E1 -19316.508,E2 -19316.508} C_VEL
LIN {X 0,Y 242.016,Z 289.965,A -85,B 0,C 180,E1 -19320.597,E2 -19320.597} C_VEL
LIN {X 0,Y 242.071,Z 289.956,A -85,B 0,C 180,E1 -19324.183,E2 -19324.183} C_VEL
LIN {X 0,Y 242.055,Z 289.958,A -85,B 0,C 180,E1 -19328.298,E2 -19328.298} C_VEL
LIN {X 0,Y 242.166,Z 289.941,A -85,B 0,C 180,E1 -19333.278,E2 -19333.278} C_VEL
LIN {X 0,Y 242.184,Z 289.944,A -85,B 0,C 180,E1 -19338.28,E2 -19338.28} C_VEL
LIN {X 0,Y 242.388,Z 289.915,A -85,B 0,C 180,E1 -19341.664,E2 -19341.664} C_VEL
LIN {X 0,Y 242.236,Z 289.933,A -85,B 0,C 180,E1 -19345.007,E2 -19345.007} C_VEL
LIN {X 0,Y 242.634,Z 289.886,A -85,B 0,C 180,E1 -19348.34,E2 -19348.34} C_VEL
LIN {X 0,Y 242.636,Z 289.884,A -85,B 0,C 180,E1 -19351.66,E2 -19351.66} C_VEL
LIN {X 0,Y 242.41,Z 289.912,A -85,B 0,C 180,E1 -19356.66,E2 -19356.66} C_VEL
LIN {X 0,Y 242.271,Z 289.931,A -85,B 0,C 180,E1 -19360.024,E2 -19360.024} C_VEL
LIN {X 0,Y 242.17,Z 289.943,A -85,B 0,C 180,E1 -19365.141,E2 -19365.141} C_VEL
LIN {X 0,Y 242.083,Z 289.951,A -85,B 0,C 180,E1 -19368.624,E2 -19368.624} C_VEL
LIN {X 0,Y 242.053,Z 289.957,A -85,B 0,C 180,E1 -19372.176,E2 -19372.176} C_VEL
LIN {X 0,Y 242.07,Z 289.954,A -85,B 0,C 180,E1 -19375.838,E2 -19375.838} C_VEL
LIN {X 0,Y 242.01,Z 289.964,A -85,B 0,C 180,E1 -19379.583,E2 -19379.583} C_VEL
LIN {X 0,Y 241.983,Z 289.965,A -85,B 0,C 180,E1 -19383.493,E2 -19383.493} C_VEL
LIN {X 0,Y 241.986,Z 289.966,A -85,B 0,C 180,E1 -19387.583,E2 -19387.583} C_VEL
LIN {X 0,Y 241.915,Z 289.972,A -85,B 0,C 180,E1 -19391.928,E2 -19391.928} C_VEL
LIN {X 0,Y 241.928,Z 289.974,A -85,B 0,C 180,E1 -19396.573,E2 -19396.573} C_VEL
LIN {X 0,Y 241.959,Z 289.967,A -85,B 0,C 180,E1 -19400.281,E2 -19400.281} C_VEL
LIN {X 0,Y 241.984,Z 289.967,A -85,B 0,C 180,E1 -19404.488,E2 -19404.488} C_VEL
LIN {X 0,Y 241.977,Z 289.968,A -85,B 0,C 180,E1 -19408.48,E2 -19408.48} C_VEL
LIN {X 0,Y 242.006,Z 289.964,A -85,B 0,C 180,E1 -19412.312,E2 -19412.312} C_VEL
LIN {X 0,Y 242.06,Z 289.956,A -85,B 0,C 180,E1 -19416.016,E2 -19416.016} C_VEL
LIN {X 0,Y 242.041,Z 289.958,A -85,B 0,C 180,E1 -19419.608,E2 -19419.608} C_VEL
LIN {X 0,Y 242.167,Z 289.942,A -85,B 0,C 180,E1 -19423.278,E2 -19423.278} C_VEL
LIN {X 0,Y 242.184,Z 289.944,A -85,B 0,C 180,E1 -19428.279,E2 -19428.279} C_VEL
LIN {X 0,Y 242.388,Z 289.915,A -85,B 0,C 180,E1 -19431.664,E2 -19431.664} C_VEL
LIN {X 0,Y 242.242,Z 289.932,A -85,B 0,C 180,E1 -19435.006,E2 -19435.006} C_VEL
LIN {X 0,Y 242.637,Z 289.886,A -85,B 0,C 180,E1 -19438.34,E2 -19438.34} C_VEL
LIN {X 0,Y 242.637,Z 289.884,A -85,B 0,C 180,E1 -19441.659,E2 -19441.659} C_VEL
LIN {X 0,Y 242.407,Z 289.913,A -85,B 0,C 180,E1 -19446.659,E2 -19446.659} C_VEL
LIN {X 0,Y 242.27,Z 289.93,A -85,B 0,C 180,E1 -19450.023,E2 -19450.023} C_VEL
LIN {X 0,Y 242.17,Z 289.943,A -85,B 0,C 180,E1 -19455.14,E2 -19455.14} C_VEL
LIN {X 0,Y 242.076,Z 289.952,A -85,B 0,C 180,E1 -19458.623,E2 -19458.623} C_VEL
LIN {X 0,Y 242.009,Z 289.964,A -85,B 0,C 180,E1 -19462.18,E2 -19462.18} C_VEL
LIN {X 0,Y 242.051,Z 290.01,A -85,B 0,C 180,E1 -19466.281,E2 -19466.281} C_VEL
LIN {X 0,Y 242.472,Z 292.954,A -85,B 0,C 180,E1 -19469.593,E2 -19469.593} C_VEL
LIN {X 0,Y 243.011,Z 296.442,A -85,B 0,C 180,E1 -19473.332,E2 -19473.332} C_VEL
LIN {X 0,Y 243.672,Z 300.309,A -85,B 0,C 180,E1 -19477.278,E2 -19477.278} C_VEL
LIN {X 0,Y 244.66,Z 304.837,A -85,B 0,C 180,E1 -19481.68,E2 -19481.68} C_VEL
LIN {X 0,Y 245.221,Z 307.591,A -85,B 0,C 180,E1 -19484.233,E2 -19484.233} C_VEL
LIN {X 0,Y 245.477,Z 310.357,A -85,B 0,C 180,E1 -19486.702,E2 -19486.702} C_VEL
LIN {X 0,Y 245.242,Z 312.885,A -85,B 0,C 180,E1 -19488.859,E2 -19488.859} C_VEL
LIN {X 0,Y 244.843,Z 314.558,A -85,B 0,C 180,E1 -19489.649,E2 -19489.649} C_VEL
LIN {X 0,Y 244.269,Z 317.145,A -85,B 0,C 180,E1 -19490.298,E2 -19490.298} C_VEL
LIN {X 0,Y 243.308,Z 322.047,A -85,B 0,C 180,E1 -19491.045,E2 -19491.045} C_VEL
LIN {X 0,Y 242.469,Z 327.901,A -85,B 0,C 180,E1 -19491.6,E2 -19491.6} C_VEL
LIN {X 0,Y 242.202,Z 335.907,A -85,B 0,C 180,E1 -19492.258,E2 -19492.258} C_VEL
LIN {X 0,Y 242.619,Z 339.644,A -85,B 0,C 180,E1 -19492.639,E2 -19492.639} C_VEL
LIN {X 0,Y 245.665,Z 356.762,A -85,B 0,C 180,E1 -19494.693,E2 -19494.693} C_VEL
LIN {X 0,Y 248.083,Z 372.24,A -85,B 0,C 180,E1 -19496.843,E2 -19496.843} C_VEL
LIN {X 0,Y 249.687,Z 383.747,A -85,B 0,C 180,E1 -19498.651,E2 -19498.651} C_VEL
LIN {X 0,Y 249.421,Z 386.47,A -85,B 0,C 180,E1 -19499.069,E2 -19499.069} C_VEL
LIN {X 0,Y 246.189,Z 399.491,A -85,B 0,C 180,E1 -19501.201,E2 -19501.201} C_VEL
LIN {X 0,Y 243.152,Z 411.717,A -85,B 0,C 180,E1 -19503.638,E2 -19503.638} C_VEL
LIN {X 0,Y 240.383,Z 422.774,A -85,B 0,C 180,E1 -19506.296,E2 -19506.296} C_VEL
LIN {X 0,Y 237.95,Z 432.914,A -85,B 0,C 180,E1 -19509.241,E2 -19509.241} C_VEL
LIN {X 0,Y 235.988,Z 441.77,A -85,B 0,C 180,E1 -19512.362,E2 -19512.362} C_VEL
LIN {X 0,Y 234.686,Z 448.566,A -85,B 0,C 180,E1 -19515.253,E2 -19515.253} C_VEL
LIN {X 0,Y 233.653,Z 455.139,A -85,B 0,C 180,E1 -19518.725,E2 -19518.725} C_VEL
LIN {X 0,Y 233.251,Z 460.254,A -85,B 0,C 180,E1 -19522.207,E2 -19522.207} C_VEL
LIN {X 0,Y 233.201,Z 463.14,A -85,B 0,C 180,E1 -19524.813,E2 -19524.813} C_VEL
LIN {X 0,Y 233.017,Z 465.856,A -85,B 0,C 180,E1 -19528.272,E2 -19528.272} C_VEL
LIN {X 0,Y 233.062,Z 466.761,A -85,B 0,C 180,E1 -19530,E2 -19530} C_VEL
LIN {X 0,Y 232.967,Z 467.589,A -85,B 0,C 180,E1 -19533.459,E2 -19533.459} C_VEL
LIN {X 0,Y 232.892,Z 467.276,A -85,B 0,C 180,E1 -19536.933,E2 -19536.933} C_VEL
LIN {X 0,Y 233.237,Z 465.933,A -85,B 0,C 180,E1 -19540.416,E2 -19540.416} C_VEL
LIN {X 0,Y 234.271,Z 463.544,A -85,B 0,C 180,E1 -19543.886,E2 -19543.886} C_VEL
LIN {X 0,Y 236.421,Z 459.471,A -85,B 0,C 180,E1 -19547.965,E2 -19547.965} C_VEL
LIN {X 0,Y 239.421,Z 454.697,A -85,B 0,C 180,E1 -19551.526,E2 -19551.526} C_VEL
LIN {X 0,Y 244.118,Z 447.743,A -85,B 0,C 180,E1 -19555.585,E2 -19555.585} C_VEL
LIN {X 0,Y 248.95,Z 441.161,A -85,B 0,C 180,E1 -19558.68,E2 -19558.68} C_VEL
LIN {X 0,Y 257.168,Z 430.474,A -85,B 0,C 180,E1 -19562.666,E2 -19562.666} C_VEL
LIN {X 0,Y 265.176,Z 420.356,A -85,B 0,C 180,E1 -19565.667,E2 -19565.667} C_VEL
LIN {X 0,Y 273.253,Z 410.24,A -85,B 0,C 180,E1 -19568.118,E2 -19568.118} C_VEL
LIN {X 0,Y 276.488,Z 406.121,A -85,B 0,C 180,E1 -19568.985,E2 -19568.985} C_VEL
LIN {X 0,Y 281.67,Z 398.628,A -85,B 0,C 180,E1 -19571.003,E2 -19571.003} C_VEL
LIN {X 0,Y 283.608,Z 395.63,A -85,B 0,C 180,E1 -19571.996,E2 -19571.996} C_VEL
LIN {X 0,Y 285.828,Z 392.191,A -85,B 0,C 180,E1 -19573.51,E2 -19573.51} C_VEL
LIN {X 0,Y 287.218,Z 390.233,A -85,B 0,C 180,E1 -19574.797,E2 -19574.797} C_VEL
LIN {X 0,Y 288.029,Z 389.622,A -85,B 0,C 180,E1 -19577.055,E2 -19577.055} C_VEL
LIN {X 0,Y 285.334,Z 392.873,A -85,B 0,C 180,E1 -19577.794,E2 -19577.794} C_VEL
LIN {X 0,Y 275.618,Z 403.978,A -85,B 0,C 180,E1 -19580.396,E2 -19580.396} C_VEL
LIN {X 0,Y 267.881,Z 412.515,A -85,B 0,C 180,E1 -19582.885,E2 -19582.885} C_VEL
LIN {X 0,Y 260.966,Z 419.943,A -85,B 0,C 180,E1 -19585.56,E2 -19585.56} C_VEL
LIN {X 0,Y 253.442,Z 427.721,A -85,B 0,C 180,E1 -19589.137,E2 -19589.137} C_VEL
LIN {X 0,Y 247.142,Z 433.896,A -85,B 0,C 180,E1 -19592.936,E2 -19592.936} C_VEL
LIN {X 0,Y 243.08,Z 437.639,A -85,B 0,C 180,E1 -19596.124,E2 -19596.124} C_VEL
LIN {X 0,Y 239.062,Z 440.856,A -85,B 0,C 180,E1 -19600.178,E2 -19600.178} C_VEL
LIN {X 0,Y 237.169,Z 442.09,A -85,B 0,C 180,E1 -19602.763,E2 -19602.763} C_VEL
LIN {X 0,Y 235.251,Z 442.7,A -85,B 0,C 180,E1 -19606.173,E2 -19606.173} C_VEL
LIN {X 0,Y 234.039,Z 442.219,A -85,B 0,C 180,E1 -19609.62,E2 -19609.62} C_VEL
LIN {X 0,Y 233.387,Z 440.628,A -85,B 0,C 180,E1 -19613.082,E2 -19613.082} C_VEL
LIN {X 0,Y 233.134,Z 437.896,A -85,B 0,C 180,E1 -19616.544,E2 -19616.544} C_VEL
LIN {X 0,Y 233.095,Z 433.927,A -85,B 0,C 180,E1 -19620,E2 -19620} C_VEL
LIN {X 0,Y 233.433,Z 428.657,A -85,B 0,C 180,E1 -19623.453,E2 -19623.453} C_VEL
LIN {X 0,Y 234.008,Z 423.735,A -85,B 0,C 180,E1 -19626.034,E2 -19626.034} C_VEL
LIN {X 0,Y 234.871,Z 415.39,A -85,B 0,C 180,E1 -19629.641,E2 -19629.641} C_VEL
LIN {X 0,Y 236.275,Z 406.139,A -85,B 0,C 180,E1 -19632.891,E2 -19632.891} C_VEL
LIN {X 0,Y 238.071,Z 396.002,A -85,B 0,C 180,E1 -19635.847,E2 -19635.847} C_VEL
LIN {X 0,Y 240.22,Z 383.927,A -85,B 0,C 180,E1 -19638.774,E2 -19638.774} C_VEL
LIN {X 0,Y 242.747,Z 370.495,A -85,B 0,C 180,E1 -19641.44,E2 -19641.44} C_VEL
LIN {X 0,Y 245.247,Z 355.666,A -85,B 0,C 180,E1 -19643.878,E2 -19643.878} C_VEL
LIN {X 0,Y 247.728,Z 340.885,A -85,B 0,C 180,E1 -19645.861,E2 -19645.861} C_VEL
LIN {X 0,Y 248.041,Z 339.305,A -85,B 0,C 180,E1 -19646.052,E2 -19646.052} C_VEL
LIN {X 0,Y 246.501,Z 331.4,A -85,B 0,C 180,E1 -19647.141,E2 -19647.141} C_VEL
LIN {X 0,Y 243.02,Z 317.113,A -85,B 0,C 180,E1 -19648.977,E2 -19648.977} C_VEL
LIN {X 0,Y 239.956,Z 306.56,A -85,B 0,C 180,E1 -19650.227,E2 -19650.227} C_VEL
LIN {X 0,Y 234.755,Z 291.628,A -85,B 0,C 180,E1 -19651.886,E2 -19651.886} C_VEL
LIN {X 0,Y 234.639,Z 290.882,A -85,B 0,C 180,E1 -19651.969,E2 -19651.969} C_VEL
LIN {X 0,Y 234.885,Z 290.854,A -85,B 0,C 180,E1 -19656.758,E2 -19656.758} C_VEL
LIN {X 0,Y 234.914,Z 290.852,A -85,B 0,C 180,E1 -19658.935,E2 -19658.935} C_VEL
LIN {X 0,Y 234.881,Z 290.853,A -85,B 0,C 180,E1 -19663.488,E2 -19663.488} C_VEL
LIN {X 0,Y 234.881,Z 290.853,A -85,B 0,C 180,E1 -19666.512,E2 -19666.512} C_VEL
LIN {X 0,Y 234.921,Z 290.848,A -85,B 0,C 180,E1 -19671.079,E2 -19671.079} C_VEL
LIN {X 0,Y 234.93,Z 290.845,A -85,B 0,C 180,E1 -19675.362,E2 -19675.362} C_VEL
LIN {X 0,Y 234.925,Z 290.845,A -85,B 0,C 180,E1 -19679.431,E2 -19679.431} C_VEL
LIN {X 0,Y 234.997,Z 290.836,A -85,B 0,C 180,E1 -19683.794,E2 -19683.794} C_VEL
LIN {X 0,Y 235.013,Z 290.834,A -85,B 0,C 180,E1 -19688.97,E2 -19688.97} C_VEL
LIN {X 0,Y 235.099,Z 290.822,A -85,B 0,C 180,E1 -19693.06,E2 -19693.06} C_VEL
LIN {X 0,Y 235.118,Z 290.822,A -85,B 0,C 180,E1 -19697.922,E2 -19697.922} C_VEL
LIN {X 0,Y 235.322,Z 290.795,A -85,B 0,C 180,E1 -19701.412,E2 -19701.412} C_VEL
LIN {X 0,Y 235.357,Z 290.788,A -85,B 0,C 180,E1 -19703.14,E2 -19703.14} C_VEL
LIN {X 0,Y 235.593,Z 290.763,A -85,B 0,C 180,E1 -19708.291,E2 -19708.291} C_VEL
LIN {X 0,Y 235.596,Z 290.761,A -85,B 0,C 180,E1 -19711.709,E2 -19711.709} C_VEL
LIN {X 0,Y 235.361,Z 290.79,A -85,B 0,C 180,E1 -19716.86,E2 -19716.86} C_VEL
LIN {X 0,Y 235.217,Z 290.807,A -85,B 0,C 180,E1 -19720.328,E2 -19720.328} C_VEL
LIN {X 0,Y 235.117,Z 290.824,A -85,B 0,C 180,E1 -19725.606,E2 -19725.606} C_VEL
LIN {X 0,Y 235.023,Z 290.832,A -85,B 0,C 180,E1 -19729.205,E2 -19729.205} C_VEL
LIN {X 0,Y 234.984,Z 290.838,A -85,B 0,C 180,E1 -19732.881,E2 -19732.881} C_VEL
LIN {X 0,Y 234.971,Z 290.837,A -85,B 0,C 180,E1 -19736.657,E2 -19736.657} C_VEL
LIN {X 0,Y 234.925,Z 290.845,A -85,B 0,C 180,E1 -19740.569,E2 -19740.569} C_VEL
LIN {X 0,Y 234.929,Z 290.842,A -85,B 0,C 180,E1 -19744.639,E2 -19744.639} C_VEL
LIN {X 0,Y 234.914,Z 290.849,A -85,B 0,C 180,E1 -19748.935,E2 -19748.935} C_VEL
LIN {X 0,Y 234.866,Z 290.852,A -85,B 0,C 180,E1 -19753.491,E2 -19753.491} C_VEL
LIN {X 0,Y 234.881,Z 290.852,A -85,B 0,C 180,E1 -19756.512,E2 -19756.512} C_VEL
LIN {X 0,Y 234.922,Z 290.846,A -85,B 0,C 180,E1 -19761.079,E2 -19761.079} C_VEL
LIN {X 0,Y 234.93,Z 290.845,A -85,B 0,C 180,E1 -19765.361,E2 -19765.361} C_VEL
LIN {X 0,Y 234.926,Z 290.843,A -85,B 0,C 180,E1 -19769.431,E2 -19769.431} C_VEL
LIN {X 0,Y 234.997,Z 290.836,A -85,B 0,C 180,E1 -19773.794,E2 -19773.794} C_VEL
LIN {X 0,Y 235.015,Z 290.834,A -85,B 0,C 180,E1 -19778.97,E2 -19778.97} C_VEL
LIN {X 0,Y 235.1,Z 290.823,A -85,B 0,C 180,E1 -19783.059,E2 -19783.059} C_VEL
LIN {X 0,Y 235.118,Z 290.822,A -85,B 0,C 180,E1 -19787.922,E2 -19787.922} C_VEL
LIN {X 0,Y 235.322,Z 290.795,A -85,B 0,C 180,E1 -19791.412,E2 -19791.412} C_VEL
LIN {X 0,Y 235.358,Z 290.788,A -85,B 0,C 180,E1 -19793.14,E2 -19793.14} C_VEL
LIN {X 0,Y 235.596,Z 290.763,A -85,B 0,C 180,E1 -19798.29,E2 -19798.29} C_VEL
LIN {X 0,Y 235.597,Z 290.762,A -85,B 0,C 180,E1 -19801.709,E2 -19801.709} C_VEL
LIN {X 0,Y 235.359,Z 290.791,A -85,B 0,C 180,E1 -19806.86,E2 -19806.86} C_VEL
LIN {X 0,Y 235.217,Z 290.807,A -85,B 0,C 180,E1 -19810.327,E2 -19810.327} C_VEL
LIN {X 0,Y 235.117,Z 290.825,A -85,B 0,C 180,E1 -19815.606,E2 -19815.606} C_VEL
LIN {X 0,Y 235.012,Z 290.834,A -85,B 0,C 180,E1 -19819.205,E2 -19819.205} C_VEL
LIN {X 0,Y 234.95,Z 290.843,A -85,B 0,C 180,E1 -19822.884,E2 -19822.884} C_VEL
LIN {X 0,Y 235.032,Z 290.968,A -85,B 0,C 180,E1 -19826.03,E2 -19826.03} C_VEL
LIN {X 0,Y 235.581,Z 294.849,A -85,B 0,C 180,E1 -19830.474,E2 -19830.474} C_VEL
LIN {X 0,Y 236.136,Z 298.507,A -85,B 0,C 180,E1 -19834.436,E2 -19834.436} C_VEL
LIN {X 0,Y 236.909,Z 302.486,A -85,B 0,C 180,E1 -19838.533,E2 -19838.533} C_VEL
LIN {X 0,Y 237.871,Z 306.849,A -85,B 0,C 180,E1 -19842.808,E2 -19842.808} C_VEL
LIN {X 0,Y 238.387,Z 310.507,A -85,B 0,C 180,E1 -19846.211,E2 -19846.211} C_VEL
LIN {X 0,Y 238.177,Z 313.341,A -85,B 0,C 180,E1 -19848.721,E2 -19848.721} C_VEL
LIN {X 0,Y 237.766,Z 315.106,A -85,B 0,C 180,E1 -19850.221,E2 -19850.221} C_VEL
LIN {X 0,Y 241.414,Z 333.624,A -85,B 0,C 180,E1 -19851.983,E2 -19851.983} C_VEL
LIN {X 0,Y 242.619,Z 339.644,A -85,B 0,C 180,E1 -19852.639,E2 -19852.639} C_VEL
LIN {X 0,Y 242.994,Z 345.082,A -85,B 0,C 180,E1 -19853.196,E2 -19853.196} C_VEL
LIN {X 0,Y 241.678,Z 354.258,A -85,B 0,C 180,E1 -19854.074,E2 -19854.074} C_VEL
LIN {X 0,Y 240.254,Z 363.21,A -85,B 0,C 180,E1 -19855.045,E2 -19855.045} C_VEL
LIN {X 0,Y 240.445,Z 368.284,A -85,B 0,C 180,E1 -19855.742,E2 -19855.742} C_VEL
LIN {X 0,Y 242.487,Z 382.818,A -85,B 0,C 180,E1 -19858.056,E2 -19858.056} C_VEL
LIN {X 0,Y 242.674,Z 385.959,A -85,B 0,C 180,E1 -19858.581,E2 -19858.581} C_VEL
LIN {X 0,Y 239.355,Z 399.02,A -85,B 0,C 180,E1 -19860.781,E2 -19860.781} C_VEL
LIN {X 0,Y 236.481,Z 410.307,A -85,B 0,C 180,E1 -19863.071,E2 -19863.071} C_VEL
LIN {X 0,Y 233.79,Z 420.68,A -85,B 0,C 180,E1 -19865.585,E2 -19865.585} C_VEL
LIN {X 0,Y 231.229,Z 431.053,A -85,B 0,C 180,E1 -19868.609,E2 -19868.609} C_VEL
LIN {X 0,Y 229.006,Z 440.879,A -85,B 0,C 180,E1 -19872.128,E2 -19872.128} C_VEL
LIN {X 0,Y 227.423,Z 448.878,A -85,B 0,C 180,E1 -19875.687,E2 -19875.687} C_VEL
LIN {X 0,Y 226.504,Z 455.258,A -85,B 0,C 180,E1 -19879.271,E2 -19879.271} C_VEL
LIN {X 0,Y 226.171,Z 460.198,A -85,B 0,C 180,E1 -19882.86,E2 -19882.86} C_VEL
LIN {X 0,Y 226.144,Z 462.155,A -85,B 0,C 180,E1 -19884.65,E2 -19884.65} C_VEL
LIN {X 0,Y 225.96,Z 465.004,A -85,B 0,C 180,E1 -19888.218,E2 -19888.218} C_VEL
LIN {X 0,Y 226.02,Z 465.96,A -85,B 0,C 180,E1 -19890,E2 -19890} C_VEL
LIN {X 0,Y 225.9,Z 466.947,A -85,B 0,C 180,E1 -19893.567,E2 -19893.567} C_VEL
LIN {X 0,Y 225.81,Z 466.83,A -85,B 0,C 180,E1 -19897.152,E2 -19897.152} C_VEL
LIN {X 0,Y 226.194,Z 465.632,A -85,B 0,C 180,E1 -19900.744,E2 -19900.744} C_VEL
LIN {X 0,Y 227.321,Z 463.446,A -85,B 0,C 180,E1 -19904.32,E2 -19904.32} C_VEL
LIN {X 0,Y 229.459,Z 459.902,A -85,B 0,C 180,E1 -19908.291,E2 -19908.291} C_VEL
LIN {X 0,Y 232.807,Z 455.193,A -85,B 0,C 180,E1 -19912.17,E2 -19912.17} C_VEL
LIN {X 0,Y 237.773,Z 448.631,A -85,B 0,C 180,E1 -19916.319,E2 -19916.319} C_VEL
LIN {X 0,Y 243.595,Z 441.465,A -85,B 0,C 180,E1 -19919.876,E2 -19919.876} C_VEL
LIN {X 0,Y 252.287,Z 431.322,A -85,B 0,C 180,E1 -19923.859,E2 -19923.859} C_VEL
LIN {X 0,Y 260.735,Z 421.64,A -85,B 0,C 180,E1 -19926.851,E2 -19926.851} C_VEL
LIN {X 0,Y 270.299,Z 410.694,A -85,B 0,C 180,E1 -19929.57,E2 -19929.57} C_VEL
LIN {X 0,Y 273.392,Z 406.956,A -85,B 0,C 180,E1 -19930.474,E2 -19930.474} C_VEL
LIN {X 0,Y 277.181,Z 402.112,A -85,B 0,C 180,E1 -19931.871,E2 -19931.871} C_VEL
LIN {X 0,Y 279.909,Z 398.426,A -85,B 0,C 180,E1 -19933.27,E2 -19933.27} C_VEL
LIN {X 0,Y 281.498,Z 396.376,A -85,B 0,C 180,E1 -19934.352,E2 -19934.352} C_VEL
LIN {X 0,Y 282.778,Z 394.913,A -85,B 0,C 180,E1 -19936.117,E2 -19936.117} C_VEL
LIN {X 0,Y 281.527,Z 396.281,A -85,B 0,C 180,E1 -19936.785,E2 -19936.785} C_VEL
LIN {X 0,Y 270.756,Z 407.459,A -85,B 0,C 180,E1 -19939.54,E2 -19939.54} C_VEL
LIN {X 0,Y 260.834,Z 417.309,A -85,B 0,C 180,E1 -19942.682,E2 -19942.682} C_VEL
LIN {X 0,Y 252.178,Z 425.508,A -85,B 0,C 180,E1 -19946.125,E2 -19946.125} C_VEL
LIN {X 0,Y 244.841,Z 432.201,A -85,B 0,C 180,E1 -19949.846,E2 -19949.846} C_VEL
LIN {X 0,Y 238.735,Z 437.368,A -85,B 0,C 180,E1 -19953.796,E2 -19953.796} C_VEL
LIN {X 0,Y 234.811,Z 440.317,A -85,B 0,C 180,E1 -19957.102,E2 -19957.102} C_VEL
LIN {X 0,Y 231.665,Z 442.296,A -85,B 0,C 180,E1 -19960.507,E2 -19960.507} C_VEL
LIN {X 0,Y 229.222,Z 443.284,A -85,B 0,C 180,E1 -19963.982,E2 -19963.982} C_VEL
LIN {X 0,Y 227.613,Z 443.179,A -85,B 0,C 180,E1 -19967.518,E2 -19967.518} C_VEL
LIN {X 0,Y 226.603,Z 441.956,A -85,B 0,C 180,E1 -19971.079,E2 -19971.079} C_VEL
LIN {X 0,Y 226.134,Z 439.618,A -85,B 0,C 180,E1 -19974.651,E2 -19974.651} C_VEL
LIN {X 0,Y 226.039,Z 436.113,A -85,B 0,C 180,E1 -19978.219,E2 -19978.219} C_VEL
LIN {X 0,Y 226.113,Z 431.348,A -85,B 0,C 180,E1 -19981.782,E2 -19981.782} C_VEL
LIN {X 0,Y 226.728,Z 425.199,A -85,B 0,C 180,E1 -19985.336,E2 -19985.336} C_VEL
LIN {X 0,Y 227.513,Z 417.535,A -85,B 0,C 180,E1 -19988.886,E2 -19988.886} C_VEL
LIN {X 0,Y 228.663,Z 409.408,A -85,B 0,C 180,E1 -19991.974,E2 -19991.974} C_VEL
LIN {X 0,Y 230.36,Z 399.751,A -85,B 0,C 180,E1 -19995.03,E2 -19995.03} C_VEL
LIN {X 0,Y 232.408,Z 388.296,A -85,B 0,C 180,E1 -19998.057,E2 -19998.057} C_VEL
LIN {X 0,Y 234.738,Z 375.707,A -85,B 0,C 180,E1 -20000.827,E2 -20000.827} C_VEL
LIN {X 0,Y 237.065,Z 363.541,A -85,B 0,C 180,E1 -20003.068,E2 -20003.068} C_VEL
LIN {X 0,Y 239.375,Z 349.739,A -85,B 0,C 180,E1 -20005.197,E2 -20005.197} C_VEL
LIN {X 0,Y 241.135,Z 339.512,A -85,B 0,C 180,E1 -20006.533,E2 -20006.533} C_VEL
LIN {X 0,Y 237.97,Z 325.34,A -85,B 0,C 180,E1 -20008.534,E2 -20008.534} C_VEL
LIN {X 0,Y 233.945,Z 310.419,A -85,B 0,C 180,E1 -20010.427,E2 -20010.427} C_VEL
LIN {X 0,Y 228.106,Z 293.575,A -85,B 0,C 180,E1 -20012.388,E2 -20012.388} C_VEL
LIN {X 0,Y 227.635,Z 291.755,A -85,B 0,C 180,E1 -20012.603,E2 -20012.603} C_VEL
